Fanuc TP program (LS listing): HS_oV_wD.ls

/PROG  HS_oV_wD
/ATTR
COMMENT	= "18-08-10 08:42:27";
PROG_SIZE	= 0;
DEFAULT_GROUP	= 1, 1, *, *, *;
/APPL
    ARC Welding Equipment: 1, *, *, *, *;
/MN
   1:  CALL HOME_ALL;
   1:  UFRAME_NUM = 1;
   1:  UTOOL_NUM = 3;
   1:  COL GUARD ADJUST 150;
   1:  PR[91] = PR[90];
   1:! Sicherheitspunkt;
   1:  PR[92] = PR[90];
   1:  PR[92] = PR[GP1:92,3] + 50;
   1:J PR[92];
   1:  PR[GP1:91,1] = PR[GP1:90,1] + -0.150;
   1:  PR[GP1:91,2] = PR[GP1:90,2] + 0.396;
   1:  PR[GP1:91,3] = PR[GP1:90,3] + 1.330;
   1:L PR[91] 10mm/sec CNT100;
   1:  PR[GP1:91,1] = PR[GP1:90,1] + -3.720;
   1:  PR[GP1:91,2] = PR[GP1:90,2] + 1.719;
   1:L PR[91] 10mm/sec CNT100;
   1:  PR[GP1:91,1] = PR[GP1:90,1] + -5.535;
   1:  PR[GP1:91,2] = PR[GP1:90,2] + 4.999;
   1:L PR[91] 10mm/sec CNT100;
   1:  PR[GP1:91,1] = PR[GP1:90,1] + -9.508;
   1:  PR[GP1:91,2] = PR[GP1:90,2] + 16.323;
   1:L PR[91] 10mm/sec CNT100;
   1:  PR[GP1:91,1] = PR[GP1:90,1] + -9.633;
   1:  PR[GP1:91,2] = PR[GP1:90,2] + 16.823;
   1:L PR[91] 10mm/sec CNT100;
   1:  PR[GP1:91,1] = PR[GP1:90,1] + -9.801;
   1:  PR[GP1:91,2] = PR[GP1:90,2] + 17.188;
   1:L PR[91] 10mm/sec CNT100;
   1:  PR[GP1:91,1] = PR[GP1:90,1] + -17.552;
   1:  PR[GP1:91,2] = PR[GP1:90,2] + 26.184;
   1:L PR[91] 10mm/sec CNT100;
   1:  PR[GP1:91,1] = PR[GP1:90,1] + -17.850;
   1:  PR[GP1:91,2] = PR[GP1:90,2] + 26.604;
   1:L PR[91] 10mm/sec CNT100;
   1:  PR[GP1:91,1] = PR[GP1:90,1] + -18.140;
   1:  PR[GP1:91,2] = PR[GP1:90,2] + 26.882;
   1:L PR[91] 10mm/sec CNT100;
   1:  PR[GP1:91,1] = PR[GP1:90,1] + -28.635;
   1:  PR[GP1:91,2] = PR[GP1:90,2] + 32.423;
   1:L PR[91] 10mm/sec CNT100;
   1:  PR[GP1:91,1] = PR[GP1:90,1] + -29.066;
   1:  PR[GP1:91,2] = PR[GP1:90,2] + 32.704;
   1:L PR[91] 10mm/sec CNT100;
   1:  PR[GP1:91,1] = PR[GP1:90,1] + -29.438;
   1:  PR[GP1:91,2] = PR[GP1:90,2] + 32.858;
   1:L PR[91] 10mm/sec CNT100;
   1:  PR[GP1:91,1] = PR[GP1:90,1] + -41.237;
   1:  PR[GP1:91,2] = PR[GP1:90,2] + 34.183;
   1:L PR[91] 10mm/sec CNT100;
   1:  PR[GP1:91,1] = PR[GP1:90,1] + -41.741;
   1:  PR[GP1:91,2] = PR[GP1:90,2] + 34.288;
   1:L PR[91] 10mm/sec CNT100;
   1:  PR[GP1:91,1] = PR[GP1:90,1] + -42.143;
   1:  PR[GP1:91,2] = PR[GP1:90,2] + 34.295;
   1:L PR[91] 10mm/sec CNT100;
   1:  PR[GP1:91,1] = PR[GP1:90,1] + -53.611;
   1:  PR[GP1:91,2] = PR[GP1:90,2] + 31.219;
   1:L PR[91] 10mm/sec CNT100;
   1:  PR[GP1:91,1] = PR[GP1:90,1] + -54.119;
   1:  PR[GP1:91,2] = PR[GP1:90,2] + 31.132;
   1:L PR[91] 10mm/sec CNT100;
   1:  PR[GP1:91,1] = PR[GP1:90,1] + -54.496;
   1:  PR[GP1:91,2] = PR[GP1:90,2] + 30.992;
   1:L PR[91] 10mm/sec CNT100;
   1:  PR[GP1:91,1] = PR[GP1:90,1] + -64.044;
   1:  PR[GP1:91,2] = PR[GP1:90,2] + 23.943;
   1:L PR[91] 10mm/sec CNT100;
   1:  PR[GP1:91,1] = PR[GP1:90,1] + -64.485;
   1:  PR[GP1:91,2] = PR[GP1:90,2] + 23.677;
   1:L PR[91] 10mm/sec CNT100;
   1:  PR[GP1:91,1] = PR[GP1:90,1] + -64.785;
   1:  PR[GP1:91,2] = PR[GP1:90,2] + 23.409;
   1:L PR[91] 10mm/sec CNT100;
   1:  PR[GP1:91,1] = PR[GP1:90,1] + -71.103;
   1:  PR[GP1:91,2] = PR[GP1:90,2] + 13.353;
   1:L PR[91] 10mm/sec CNT100;
   1:  PR[GP1:91,1] = PR[GP1:90,1] + -71.416;
   1:  PR[GP1:91,2] = PR[GP1:90,2] + 12.944;
   1:L PR[91] 10mm/sec CNT100;
   1:  PR[GP1:91,1] = PR[GP1:90,1] + -71.597;
   1:  PR[GP1:91,2] = PR[GP1:90,2] + 12.585;
   1:L PR[91] 10mm/sec CNT100;
   1:  PR[GP1:91,1] = PR[GP1:90,1] + -73.804;
   1:  PR[GP1:91,2] = PR[GP1:90,2] + 0.919;
   1:L PR[91] 10mm/sec CNT100;
   1:  PR[GP1:91,1] = PR[GP1:90,1] + -73.947;
   1:  PR[GP1:91,2] = PR[GP1:90,2] + 0.424;
   1:L PR[91] 10mm/sec CNT100;
   1:  PR[GP1:91,1] = PR[GP1:90,1] + -73.984;
   1:  PR[GP1:91,2] = PR[GP1:90,2] + 0.024;
   1:L PR[91] 10mm/sec CNT100;
   1:  PR[GP1:91,1] = PR[GP1:90,1] + -71.777;
   1:  PR[GP1:91,2] = PR[GP1:90,2] + -11.642;
   1:L PR[91] 10mm/sec CNT100;
   1:  PR[GP1:91,1] = PR[GP1:90,1] + -71.729;
   1:  PR[GP1:91,2] = PR[GP1:90,2] + -12.155;
   1:L PR[91] 10mm/sec CNT100;
   1:  PR[GP1:91,1] = PR[GP1:90,1] + -71.610;
   1:  PR[GP1:91,2] = PR[GP1:90,2] + -12.569;
   1:L PR[91] 10mm/sec CNT100;
   1:  PR[GP1:91,1] = PR[GP1:90,1] + -71.403;
   1:  PR[GP1:91,2] = PR[GP1:90,2] + -12.978;
   1:L PR[91] 10mm/sec CNT100;
   1:  PR[GP1:91,1] = PR[GP1:90,1] + -65.085;
   1:  PR[GP1:91,2] = PR[GP1:90,2] + -23.035;
   1:L PR[91] 10mm/sec CNT100;
   1:  PR[GP1:91,1] = PR[GP1:90,1] + -64.806;
   1:  PR[GP1:91,2] = PR[GP1:90,2] + -23.399;
   1:L PR[91] 10mm/sec CNT100;
   1:  PR[GP1:91,1] = PR[GP1:90,1] + -64.464;
   1:  PR[GP1:91,2] = PR[GP1:90,2] + -23.705;
   1:L PR[91] 10mm/sec CNT100;
   1:  PR[GP1:91,1] = PR[GP1:90,1] + -54.915;
   1:  PR[GP1:91,2] = PR[GP1:90,2] + -30.754;
   1:L PR[91] 10mm/sec CNT100;
   1:  PR[GP1:91,1] = PR[GP1:90,1] + -54.522;
   1:  PR[GP1:91,2] = PR[GP1:90,2] + -30.991;
   1:L PR[91] 10mm/sec CNT100;
   1:  PR[GP1:91,1] = PR[GP1:90,1] + -54.092;
   1:  PR[GP1:91,2] = PR[GP1:90,2] + -31.151;
   1:L PR[91] 10mm/sec CNT100;
   1:  PR[GP1:91,1] = PR[GP1:90,1] + -42.624;
   1:  PR[GP1:91,2] = PR[GP1:90,2] + -34.227;
   1:L PR[91] 10mm/sec CNT100;
   1:  PR[GP1:91,1] = PR[GP1:90,1] + -42.171;
   1:  PR[GP1:91,2] = PR[GP1:90,2] + -34.304;
   1:L PR[91] 10mm/sec CNT100;
   1:  PR[GP1:91,1] = PR[GP1:90,1] + -41.713;
   1:  PR[GP1:91,2] = PR[GP1:90,2] + -34.296;
   1:L PR[91] 10mm/sec CNT100;
   1:  PR[GP1:91,1] = PR[GP1:90,1] + -29.913;
   1:  PR[GP1:91,2] = PR[GP1:90,2] + -32.971;
   1:L PR[91] 10mm/sec CNT100;
   1:  PR[GP1:91,1] = PR[GP1:90,1] + -29.464;
   1:  PR[GP1:91,2] = PR[GP1:90,2] + -32.878;
   1:L PR[91] 10mm/sec CNT100;
   1:  PR[GP1:91,1] = PR[GP1:90,1] + -29.040;
   1:  PR[GP1:91,2] = PR[GP1:90,2] + -32.702;
   1:L PR[91] 10mm/sec CNT100;
   1:  PR[GP1:91,1] = PR[GP1:90,1] + -18.545;
   1:  PR[GP1:91,2] = PR[GP1:90,2] + -27.162;
   1:L PR[91] 10mm/sec CNT100;
   1:  PR[GP1:91,1] = PR[GP1:90,1] + -18.161;
   1:  PR[GP1:91,2] = PR[GP1:90,2] + -26.911;
   1:L PR[91] 10mm/sec CNT100;
   1:  PR[GP1:91,1] = PR[GP1:90,1] + -17.830;
   1:  PR[GP1:91,2] = PR[GP1:90,2] + -26.593;
   1:L PR[91] 10mm/sec CNT100;
   1:  PR[GP1:91,1] = PR[GP1:90,1] + -10.079;
   1:  PR[GP1:91,2] = PR[GP1:90,2] + -17.597;
   1:L PR[91] 10mm/sec CNT100;
   1:  PR[GP1:91,1] = PR[GP1:90,1] + -9.813;
   1:  PR[GP1:91,2] = PR[GP1:90,2] + -17.223;
   1:L PR[91] 10mm/sec CNT100;
   1:  PR[GP1:91,1] = PR[GP1:90,1] + -9.621;
   1:  PR[GP1:91,2] = PR[GP1:90,2] + -16.806;
   1:L PR[91] 10mm/sec CNT100;
   1:  PR[GP1:91,1] = PR[GP1:90,1] + -5.692;
   1:  PR[GP1:91,2] = PR[GP1:90,2] + -5.609;
   1:L PR[91] 10mm/sec CNT100;
   1:  PR[GP1:91,1] = PR[GP1:90,1] + -5.549;
   1:  PR[GP1:91,2] = PR[GP1:90,2] + -5.033;
   1:L PR[91] 10mm/sec CNT100;
   1:  PR[GP1:91,1] = PR[GP1:90,1] + -3.720;
   1:  PR[GP1:91,2] = PR[GP1:90,2] + -1.728;
   1:L PR[91] 10mm/sec CNT100;
   1:  PR[GP1:91,1] = PR[GP1:90,1] + -0.150;
   1:  PR[GP1:91,2] = PR[GP1:90,2] + -0.404;
   1:L PR[91] 10mm/sec CNT100;
   1:  PR[GP1:91,1] = PR[GP1:90,1] + 0.971;
   1:L PR[91] 10mm/sec CNT100;
   1:  PR[GP1:91,1] = PR[GP1:90,1] + 4.540;
   1:  PR[GP1:91,2] = PR[GP1:90,2] + -1.728;
   1:L PR[91] 10mm/sec CNT100;
   1:  PR[GP1:91,1] = PR[GP1:90,1] + 6.356;
   1:  PR[GP1:91,2] = PR[GP1:90,2] + -5.008;
   1:L PR[91] 10mm/sec CNT100;
   1:  PR[GP1:91,1] = PR[GP1:90,1] + 10.329;
   1:  PR[GP1:91,2] = PR[GP1:90,2] + -16.332;
   1:L PR[91] 10mm/sec CNT100;
   1:  PR[GP1:91,1] = PR[GP1:90,1] + 10.453;
   1:  PR[GP1:91,2] = PR[GP1:90,2] + -16.832;
   1:L PR[91] 10mm/sec CNT100;
   1:  PR[GP1:91,1] = PR[GP1:90,1] + 10.621;
   1:  PR[GP1:91,2] = PR[GP1:90,2] + -17.197;
   1:L PR[91] 10mm/sec CNT100;
   1:  PR[GP1:91,1] = PR[GP1:90,1] + 18.373;
   1:  PR[GP1:91,2] = PR[GP1:90,2] + -26.193;
   1:L PR[91] 10mm/sec CNT100;
   1:  PR[GP1:91,1] = PR[GP1:90,1] + 18.671;
   1:  PR[GP1:91,2] = PR[GP1:90,2] + -26.612;
   1:L PR[91] 10mm/sec CNT100;
   1:  PR[GP1:91,1] = PR[GP1:90,1] + 18.961;
   1:  PR[GP1:91,2] = PR[GP1:90,2] + -26.891;
   1:L PR[91] 10mm/sec CNT100;
   1:  PR[GP1:91,1] = PR[GP1:90,1] + 29.456;
   1:  PR[GP1:91,2] = PR[GP1:90,2] + -32.431;
   1:L PR[91] 10mm/sec CNT100;
   1:  PR[GP1:91,1] = PR[GP1:90,1] + 29.887;
   1:  PR[GP1:91,2] = PR[GP1:90,2] + -32.713;
   1:L PR[91] 10mm/sec CNT100;
   1:  PR[GP1:91,1] = PR[GP1:90,1] + 30.259;
   1:  PR[GP1:91,2] = PR[GP1:90,2] + -32.867;
   1:L PR[91] 10mm/sec CNT100;
   1:  PR[GP1:91,1] = PR[GP1:90,1] + 42.058;
   1:  PR[GP1:91,2] = PR[GP1:90,2] + -34.192;
   1:L PR[91] 10mm/sec CNT100;
   1:  PR[GP1:91,1] = PR[GP1:90,1] + 42.562;
   1:  PR[GP1:91,2] = PR[GP1:90,2] + -34.296;
   1:L PR[91] 10mm/sec CNT100;
   1:  PR[GP1:91,1] = PR[GP1:90,1] + 42.964;
   1:  PR[GP1:91,2] = PR[GP1:90,2] + -34.304;
   1:L PR[91] 10mm/sec CNT100;
   1:  PR[GP1:91,1] = PR[GP1:90,1] + 54.432;
   1:  PR[GP1:91,2] = PR[GP1:90,2] + -31.228;
   1:L PR[91] 10mm/sec CNT100;
   1:  PR[GP1:91,1] = PR[GP1:90,1] + 54.939;
   1:  PR[GP1:91,2] = PR[GP1:90,2] + -31.141;
   1:L PR[91] 10mm/sec CNT100;
   1:  PR[GP1:91,1] = PR[GP1:90,1] + 55.316;
   1:  PR[GP1:91,2] = PR[GP1:90,2] + -31.001;
   1:L PR[91] 10mm/sec CNT100;
   1:  PR[GP1:91,1] = PR[GP1:90,1] + 64.865;
   1:  PR[GP1:91,2] = PR[GP1:90,2] + -23.952;
   1:L PR[91] 10mm/sec CNT100;
   1:  PR[GP1:91,1] = PR[GP1:90,1] + 65.306;
   1:  PR[GP1:91,2] = PR[GP1:90,2] + -23.686;
   1:L PR[91] 10mm/sec CNT100;
   1:  PR[GP1:91,1] = PR[GP1:90,1] + 65.605;
   1:  PR[GP1:91,2] = PR[GP1:90,2] + -23.418;
   1:L PR[91] 10mm/sec CNT100;
   1:  PR[GP1:91,1] = PR[GP1:90,1] + 71.923;
   1:  PR[GP1:91,2] = PR[GP1:90,2] + -13.361;
   1:L PR[91] 10mm/sec CNT100;
   1:  PR[GP1:91,1] = PR[GP1:90,1] + 72.237;
   1:  PR[GP1:91,2] = PR[GP1:90,2] + -12.953;
   1:L PR[91] 10mm/sec CNT100;
   1:  PR[GP1:91,1] = PR[GP1:90,1] + 72.418;
   1:  PR[GP1:91,2] = PR[GP1:90,2] + -12.594;
   1:L PR[91] 10mm/sec CNT100;
   1:  PR[GP1:91,1] = PR[GP1:90,1] + 74.625;
   1:  PR[GP1:91,2] = PR[GP1:90,2] + -0.928;
   1:L PR[91] 10mm/sec CNT100;
   1:  PR[GP1:91,1] = PR[GP1:90,1] + 74.767;
   1:  PR[GP1:91,2] = PR[GP1:90,2] + -0.433;
   1:L PR[91] 10mm/sec CNT100;
   1:  PR[GP1:91,1] = PR[GP1:90,1] + 74.805;
   1:  PR[GP1:91,2] = PR[GP1:90,2] + -0.033;
   1:L PR[91] 10mm/sec CNT100;
   1:  PR[GP1:91,1] = PR[GP1:90,1] + 72.598;
   1:  PR[GP1:91,2] = PR[GP1:90,2] + 11.633;
   1:L PR[91] 10mm/sec CNT100;
   1:  PR[GP1:91,1] = PR[GP1:90,1] + 72.550;
   1:  PR[GP1:91,2] = PR[GP1:90,2] + 12.146;
   1:L PR[91] 10mm/sec CNT100;
   1:  PR[GP1:91,1] = PR[GP1:90,1] + 72.430;
   1:  PR[GP1:91,2] = PR[GP1:90,2] + 12.560;
   1:L PR[91] 10mm/sec CNT100;
   1:  PR[GP1:91,1] = PR[GP1:90,1] + 72.224;
   1:  PR[GP1:91,2] = PR[GP1:90,2] + 12.969;
   1:L PR[91] 10mm/sec CNT100;
   1:  PR[GP1:91,1] = PR[GP1:90,1] + 65.906;
   1:  PR[GP1:91,2] = PR[GP1:90,2] + 23.026;
   1:L PR[91] 10mm/sec CNT100;
   1:  PR[GP1:91,1] = PR[GP1:90,1] + 65.627;
   1:  PR[GP1:91,2] = PR[GP1:90,2] + 23.390;
   1:L PR[91] 10mm/sec CNT100;
   1:  PR[GP1:91,1] = PR[GP1:90,1] + 65.285;
   1:  PR[GP1:91,2] = PR[GP1:90,2] + 23.696;
   1:L PR[91] 10mm/sec CNT100;
   1:  PR[GP1:91,1] = PR[GP1:90,1] + 55.736;
   1:  PR[GP1:91,2] = PR[GP1:90,2] + 30.746;
   1:L PR[91] 10mm/sec CNT100;
   1:  PR[GP1:91,1] = PR[GP1:90,1] + 55.343;
   1:  PR[GP1:91,2] = PR[GP1:90,2] + 30.982;
   1:L PR[91] 10mm/sec CNT100;
   1:  PR[GP1:91,1] = PR[GP1:90,1] + 54.913;
   1:  PR[GP1:91,2] = PR[GP1:90,2] + 31.142;
   1:L PR[91] 10mm/sec CNT100;
   1:  PR[GP1:91,1] = PR[GP1:90,1] + 43.444;
   1:  PR[GP1:91,2] = PR[GP1:90,2] + 34.218;
   1:L PR[91] 10mm/sec CNT100;
   1:  PR[GP1:91,1] = PR[GP1:90,1] + 42.992;
   1:  PR[GP1:91,2] = PR[GP1:90,2] + 34.295;
   1:L PR[91] 10mm/sec CNT100;
   1:  PR[GP1:91,1] = PR[GP1:90,1] + 42.533;
   1:  PR[GP1:91,2] = PR[GP1:90,2] + 34.287;
   1:L PR[91] 10mm/sec CNT100;
   1:  PR[GP1:91,1] = PR[GP1:90,1] + 30.734;
   1:  PR[GP1:91,2] = PR[GP1:90,2] + 32.962;
   1:L PR[91] 10mm/sec CNT100;
   1:  PR[GP1:91,1] = PR[GP1:90,1] + 30.285;
   1:  PR[GP1:91,2] = PR[GP1:90,2] + 32.869;
   1:L PR[91] 10mm/sec CNT100;
   1:  PR[GP1:91,1] = PR[GP1:90,1] + 29.861;
   1:  PR[GP1:91,2] = PR[GP1:90,2] + 32.694;
   1:L PR[91] 10mm/sec CNT100;
   1:  PR[GP1:91,1] = PR[GP1:90,1] + 19.365;
   1:  PR[GP1:91,2] = PR[GP1:90,2] + 27.153;
   1:L PR[91] 10mm/sec CNT100;
   1:  PR[GP1:91,1] = PR[GP1:90,1] + 18.981;
   1:  PR[GP1:91,2] = PR[GP1:90,2] + 26.902;
   1:L PR[91] 10mm/sec CNT100;
   1:  PR[GP1:91,1] = PR[GP1:90,1] + 18.651;
   1:  PR[GP1:91,2] = PR[GP1:90,2] + 26.584;
   1:L PR[91] 10mm/sec CNT100;
   1:  PR[GP1:91,1] = PR[GP1:90,1] + 10.899;
   1:  PR[GP1:91,2] = PR[GP1:90,2] + 17.588;
   1:L PR[91] 10mm/sec CNT100;
   1:  PR[GP1:91,1] = PR[GP1:90,1] + 10.633;
   1:  PR[GP1:91,2] = PR[GP1:90,2] + 17.214;
   1:L PR[91] 10mm/sec CNT100;
   1:  PR[GP1:91,1] = PR[GP1:90,1] + 10.442;
   1:  PR[GP1:91,2] = PR[GP1:90,2] + 16.797;
   1:L PR[91] 10mm/sec CNT100;
   1:  PR[GP1:91,1] = PR[GP1:90,1] + 6.513;
   1:  PR[GP1:91,2] = PR[GP1:90,2] + 5.600;
   1:L PR[91] 10mm/sec CNT100;
   1:  PR[GP1:91,1] = PR[GP1:90,1] + 6.369;
   1:  PR[GP1:91,2] = PR[GP1:90,2] + 5.024;
   1:L PR[91] 10mm/sec CNT100;
   1:  PR[GP1:91,1] = PR[GP1:90,1] + 4.540;
   1:  PR[GP1:91,2] = PR[GP1:90,2] + 1.719;
   1:L PR[91] 10mm/sec CNT100;
   1:  PR[GP1:91,1] = PR[GP1:90,1] + 0.971;
   1:  PR[GP1:91,2] = PR[GP1:90,2] + 0.396;
   1:L PR[91] 10mm/sec CNT100;
   1:  PR[GP1:91,1] = PR[GP1:90,1] + -0.150;
   1:L PR[91] 10mm/sec CNT100;
   1:  PR[GP1:91,1] = PR[GP1:90,1] + -3.720;
   1:  PR[GP1:91,2] = PR[GP1:90,2] + 1.719;
   1:  PR[GP1:91,3] = PR[GP1:90,3] + 2.660;
   1:L PR[91] 10mm/sec CNT100;
   1:  PR[GP1:91,1] = PR[GP1:90,1] + -5.535;
   1:  PR[GP1:91,2] = PR[GP1:90,2] + 4.999;
   1:L PR[91] 10mm/sec CNT100;
   1:  PR[GP1:91,1] = PR[GP1:90,1] + -8.793;
   1:  PR[GP1:91,2] = PR[GP1:90,2] + 14.283;
   1:L PR[91] 10mm/sec CNT100;
   1:  PR[GP1:91,1] = PR[GP1:90,1] + -9.180;
   1:  PR[GP1:91,2] = PR[GP1:90,2] + 15.837;
   1:L PR[91] 10mm/sec CNT100;
   1:  PR[GP1:91,1] = PR[GP1:90,1] + -9.801;
   1:  PR[GP1:91,2] = PR[GP1:90,2] + 17.189;
   1:L PR[91] 10mm/sec CNT100;
   1:  PR[GP1:91,1] = PR[GP1:90,1] + -16.140;
   1:  PR[GP1:91,2] = PR[GP1:90,2] + 24.546;
   1:L PR[91] 10mm/sec CNT100;
   1:  PR[GP1:91,1] = PR[GP1:90,1] + -17.068;
   1:  PR[GP1:91,2] = PR[GP1:90,2] + 25.851;
   1:L PR[91] 10mm/sec CNT100;
   1:  PR[GP1:91,1] = PR[GP1:90,1] + -18.141;
   1:  PR[GP1:91,2] = PR[GP1:90,2] + 26.883;
   1:L PR[91] 10mm/sec CNT100;
   1:  PR[GP1:91,1] = PR[GP1:90,1] + -26.724;
   1:  PR[GP1:91,2] = PR[GP1:90,2] + 31.414;
   1:L PR[91] 10mm/sec CNT100;
   1:  PR[GP1:91,1] = PR[GP1:90,1] + -28.064;
   1:  PR[GP1:91,2] = PR[GP1:90,2] + 32.290;
   1:L PR[91] 10mm/sec CNT100;
   1:  PR[GP1:91,1] = PR[GP1:90,1] + -29.439;
   1:  PR[GP1:91,2] = PR[GP1:90,2] + 32.858;
   1:L PR[91] 10mm/sec CNT100;
   1:  PR[GP1:91,1] = PR[GP1:90,1] + -39.088;
   1:  PR[GP1:91,2] = PR[GP1:90,2] + 33.942;
   1:L PR[91] 10mm/sec CNT100;
   1:  PR[GP1:91,1] = PR[GP1:90,1] + -40.656;
   1:  PR[GP1:91,2] = PR[GP1:90,2] + 34.268;
   1:L PR[91] 10mm/sec CNT100;
   1:  PR[GP1:91,1] = PR[GP1:90,1] + -42.144;
   1:  PR[GP1:91,2] = PR[GP1:90,2] + 34.295;
   1:L PR[91] 10mm/sec CNT100;
   1:  PR[GP1:91,1] = PR[GP1:90,1] + -51.523;
   1:  PR[GP1:91,2] = PR[GP1:90,2] + 31.779;
   1:L PR[91] 10mm/sec CNT100;
   1:  PR[GP1:91,1] = PR[GP1:90,1] + -53.101;
   1:  PR[GP1:91,2] = PR[GP1:90,2] + 31.510;
   1:L PR[91] 10mm/sec CNT100;
   1:  PR[GP1:91,1] = PR[GP1:90,1] + -54.496;
   1:  PR[GP1:91,2] = PR[GP1:90,2] + 30.992;
   1:L PR[91] 10mm/sec CNT100;
   1:  PR[GP1:91,1] = PR[GP1:90,1] + -62.305;
   1:  PR[GP1:91,2] = PR[GP1:90,2] + 25.227;
   1:L PR[91] 10mm/sec CNT100;
   1:  PR[GP1:91,1] = PR[GP1:90,1] + -63.676;
   1:  PR[GP1:91,2] = PR[GP1:90,2] + 24.400;
   1:L PR[91] 10mm/sec CNT100;
   1:  PR[GP1:91,1] = PR[GP1:90,1] + -64.786;
   1:  PR[GP1:91,2] = PR[GP1:90,2] + 23.408;
   1:L PR[91] 10mm/sec CNT100;
   1:  PR[GP1:91,1] = PR[GP1:90,1] + -69.952;
   1:  PR[GP1:91,2] = PR[GP1:90,2] + 15.184;
   1:L PR[91] 10mm/sec CNT100;
   1:  PR[GP1:91,1] = PR[GP1:90,1] + -70.927;
   1:  PR[GP1:91,2] = PR[GP1:90,2] + 13.914;
   1:L PR[91] 10mm/sec CNT100;
   1:  PR[GP1:91,1] = PR[GP1:90,1] + -71.597;
   1:  PR[GP1:91,2] = PR[GP1:90,2] + 12.585;
   1:L PR[91] 10mm/sec CNT100;
   1:  PR[GP1:91,1] = PR[GP1:90,1] + -73.402;
   1:  PR[GP1:91,2] = PR[GP1:90,2] + 3.044;
   1:L PR[91] 10mm/sec CNT100;
   1:  PR[GP1:91,1] = PR[GP1:90,1] + -73.845;
   1:  PR[GP1:91,2] = PR[GP1:90,2] + 1.506;
   1:L PR[91] 10mm/sec CNT100;
   1:  PR[GP1:91,1] = PR[GP1:90,1] + -73.984;
   1:  PR[GP1:91,2] = PR[GP1:90,2] + 0.024;
   1:L PR[91] 10mm/sec CNT100;
   1:  PR[GP1:91,1] = PR[GP1:90,1] + -72.179;
   1:  PR[GP1:91,2] = PR[GP1:90,2] + -9.517;
   1:L PR[91] 10mm/sec CNT100;
   1:  PR[GP1:91,1] = PR[GP1:90,1] + -72.030;
   1:  PR[GP1:91,2] = PR[GP1:90,2] + -11.111;
   1:L PR[91] 10mm/sec CNT100;
   1:  PR[GP1:91,1] = PR[GP1:90,1] + -71.610;
   1:  PR[GP1:91,2] = PR[GP1:90,2] + -12.568;
   1:L PR[91] 10mm/sec CNT100;
   1:  PR[GP1:91,1] = PR[GP1:90,1] + -70.914;
   1:  PR[GP1:91,2] = PR[GP1:90,2] + -13.948;
   1:L PR[91] 10mm/sec CNT100;
   1:  PR[GP1:91,1] = PR[GP1:90,1] + -65.747;
   1:  PR[GP1:91,2] = PR[GP1:90,2] + -22.172;
   1:L PR[91] 10mm/sec CNT100;
   1:  PR[GP1:91,1] = PR[GP1:90,1] + -64.807;
   1:  PR[GP1:91,2] = PR[GP1:90,2] + -23.398;
   1:L PR[91] 10mm/sec CNT100;
   1:  PR[GP1:91,1] = PR[GP1:90,1] + -63.655;
   1:  PR[GP1:91,2] = PR[GP1:90,2] + -24.428;
   1:L PR[91] 10mm/sec CNT100;
   1:  PR[GP1:91,1] = PR[GP1:90,1] + -55.846;
   1:  PR[GP1:91,2] = PR[GP1:90,2] + -30.193;
   1:L PR[91] 10mm/sec CNT100;
   1:  PR[GP1:91,1] = PR[GP1:90,1] + -54.523;
   1:  PR[GP1:91,2] = PR[GP1:90,2] + -30.991;
   1:L PR[91] 10mm/sec CNT100;
   1:  PR[GP1:91,1] = PR[GP1:90,1] + -53.075;
   1:  PR[GP1:91,2] = PR[GP1:90,2] + -31.529;
   1:L PR[91] 10mm/sec CNT100;
   1:  PR[GP1:91,1] = PR[GP1:90,1] + -43.695;
   1:  PR[GP1:91,2] = PR[GP1:90,2] + -34.045;
   1:L PR[91] 10mm/sec CNT100;
   1:  PR[GP1:91,1] = PR[GP1:90,1] + -42.172;
   1:  PR[GP1:91,2] = PR[GP1:90,2] + -34.304;
   1:L PR[91] 10mm/sec CNT100;
   1:  PR[GP1:91,1] = PR[GP1:90,1] + -40.628;
   1:  PR[GP1:91,2] = PR[GP1:90,2] + -34.276;
   1:L PR[91] 10mm/sec CNT100;
   1:  PR[GP1:91,1] = PR[GP1:90,1] + -30.978;
   1:  PR[GP1:91,2] = PR[GP1:90,2] + -33.193;
   1:L PR[91] 10mm/sec CNT100;
   1:  PR[GP1:91,1] = PR[GP1:90,1] + -29.465;
   1:  PR[GP1:91,2] = PR[GP1:90,2] + -32.878;
   1:L PR[91] 10mm/sec CNT100;
   1:  PR[GP1:91,1] = PR[GP1:90,1] + -28.038;
   1:  PR[GP1:91,2] = PR[GP1:90,2] + -32.288;
   1:L PR[91] 10mm/sec CNT100;
   1:  PR[GP1:91,1] = PR[GP1:90,1] + -19.454;
   1:  PR[GP1:91,2] = PR[GP1:90,2] + -27.757;
   1:L PR[91] 10mm/sec CNT100;
   1:  PR[GP1:91,1] = PR[GP1:90,1] + -18.161;
   1:  PR[GP1:91,2] = PR[GP1:90,2] + -26.911;
   1:L PR[91] 10mm/sec CNT100;
   1:  PR[GP1:91,1] = PR[GP1:90,1] + -17.048;
   1:  PR[GP1:91,2] = PR[GP1:90,2] + -25.840;
   1:L PR[91] 10mm/sec CNT100;
   1:  PR[GP1:91,1] = PR[GP1:90,1] + -10.708;
   1:  PR[GP1:91,2] = PR[GP1:90,2] + -18.483;
   1:L PR[91] 10mm/sec CNT100;
   1:  PR[GP1:91,1] = PR[GP1:90,1] + -9.813;
   1:  PR[GP1:91,2] = PR[GP1:90,2] + -17.224;
   1:L PR[91] 10mm/sec CNT100;
   1:  PR[GP1:91,1] = PR[GP1:90,1] + -9.168;
   1:  PR[GP1:91,2] = PR[GP1:90,2] + -15.820;
   1:L PR[91] 10mm/sec CNT100;
   1:  PR[GP1:91,1] = PR[GP1:90,1] + -5.955;
   1:  PR[GP1:91,2] = PR[GP1:90,2] + -6.663;
   1:L PR[91] 10mm/sec CNT100;
   1:  PR[GP1:91,1] = PR[GP1:90,1] + -5.549;
   1:  PR[GP1:91,2] = PR[GP1:90,2] + -5.033;
   1:L PR[91] 10mm/sec CNT100;
   1:  PR[GP1:91,1] = PR[GP1:90,1] + -3.720;
   1:  PR[GP1:91,2] = PR[GP1:90,2] + -1.728;
   1:L PR[91] 10mm/sec CNT100;
   1:  PR[GP1:91,1] = PR[GP1:90,1] + -0.150;
   1:  PR[GP1:91,2] = PR[GP1:90,2] + -0.404;
   1:L PR[91] 10mm/sec CNT100;
   1:  PR[GP1:91,1] = PR[GP1:90,1] + 0.971;
   1:L PR[91] 10mm/sec CNT100;
   1:  PR[GP1:91,1] = PR[GP1:90,1] + 4.540;
   1:  PR[GP1:91,2] = PR[GP1:90,2] + -1.728;
   1:L PR[91] 10mm/sec CNT100;
   1:  PR[GP1:91,1] = PR[GP1:90,1] + 6.356;
   1:  PR[GP1:91,2] = PR[GP1:90,2] + -5.008;
   1:L PR[91] 10mm/sec CNT100;
   1:  PR[GP1:91,1] = PR[GP1:90,1] + 9.613;
   1:  PR[GP1:91,2] = PR[GP1:90,2] + -14.292;
   1:L PR[91] 10mm/sec CNT100;
   1:  PR[GP1:91,1] = PR[GP1:90,1] + 10.000;
   1:  PR[GP1:91,2] = PR[GP1:90,2] + -15.846;
   1:L PR[91] 10mm/sec CNT100;
   1:  PR[GP1:91,1] = PR[GP1:90,1] + 10.622;
   1:  PR[GP1:91,2] = PR[GP1:90,2] + -17.198;
   1:L PR[91] 10mm/sec CNT100;
   1:  PR[GP1:91,1] = PR[GP1:90,1] + 16.961;
   1:  PR[GP1:91,2] = PR[GP1:90,2] + -24.555;
   1:L PR[91] 10mm/sec CNT100;
   1:  PR[GP1:91,1] = PR[GP1:90,1] + 17.889;
   1:  PR[GP1:91,2] = PR[GP1:90,2] + -25.860;
   1:L PR[91] 10mm/sec CNT100;
   1:  PR[GP1:91,1] = PR[GP1:90,1] + 18.961;
   1:  PR[GP1:91,2] = PR[GP1:90,2] + -26.892;
   1:L PR[91] 10mm/sec CNT100;
   1:  PR[GP1:91,1] = PR[GP1:90,1] + 27.544;
   1:  PR[GP1:91,2] = PR[GP1:90,2] + -31.422;
   1:L PR[91] 10mm/sec CNT100;
   1:  PR[GP1:91,1] = PR[GP1:90,1] + 28.884;
   1:  PR[GP1:91,2] = PR[GP1:90,2] + -32.298;
   1:L PR[91] 10mm/sec CNT100;
   1:  PR[GP1:91,1] = PR[GP1:90,1] + 30.260;
   1:  PR[GP1:91,2] = PR[GP1:90,2] + -32.867;
   1:L PR[91] 10mm/sec CNT100;
   1:  PR[GP1:91,1] = PR[GP1:90,1] + 39.909;
   1:  PR[GP1:91,2] = PR[GP1:90,2] + -33.951;
   1:L PR[91] 10mm/sec CNT100;
   1:  PR[GP1:91,1] = PR[GP1:90,1] + 41.477;
   1:  PR[GP1:91,2] = PR[GP1:90,2] + -34.277;
   1:L PR[91] 10mm/sec CNT100;
   1:  PR[GP1:91,1] = PR[GP1:90,1] + 42.965;
   1:  PR[GP1:91,2] = PR[GP1:90,2] + -34.304;
   1:L PR[91] 10mm/sec CNT100;
   1:  PR[GP1:91,1] = PR[GP1:90,1] + 52.343;
   1:  PR[GP1:91,2] = PR[GP1:90,2] + -31.788;
   1:L PR[91] 10mm/sec CNT100;
   1:  PR[GP1:91,1] = PR[GP1:90,1] + 53.922;
   1:  PR[GP1:91,2] = PR[GP1:90,2] + -31.519;
   1:L PR[91] 10mm/sec CNT100;
   1:  PR[GP1:91,1] = PR[GP1:90,1] + 55.317;
   1:  PR[GP1:91,2] = PR[GP1:90,2] + -31.001;
   1:L PR[91] 10mm/sec CNT100;
   1:  PR[GP1:91,1] = PR[GP1:90,1] + 63.126;
   1:  PR[GP1:91,2] = PR[GP1:90,2] + -25.236;
   1:L PR[91] 10mm/sec CNT100;
   1:  PR[GP1:91,1] = PR[GP1:90,1] + 64.497;
   1:  PR[GP1:91,2] = PR[GP1:90,2] + -24.409;
   1:L PR[91] 10mm/sec CNT100;
   1:  PR[GP1:91,1] = PR[GP1:90,1] + 65.606;
   1:  PR[GP1:91,2] = PR[GP1:90,2] + -23.417;
   1:L PR[91] 10mm/sec CNT100;
   1:  PR[GP1:91,1] = PR[GP1:90,1] + 70.773;
   1:  PR[GP1:91,2] = PR[GP1:90,2] + -15.193;
   1:L PR[91] 10mm/sec CNT100;
   1:  PR[GP1:91,1] = PR[GP1:90,1] + 71.747;
   1:  PR[GP1:91,2] = PR[GP1:90,2] + -13.922;
   1:L PR[91] 10mm/sec CNT100;
   1:  PR[GP1:91,1] = PR[GP1:90,1] + 72.418;
   1:  PR[GP1:91,2] = PR[GP1:90,2] + -12.594;
   1:L PR[91] 10mm/sec CNT100;
   1:  PR[GP1:91,1] = PR[GP1:90,1] + 74.223;
   1:  PR[GP1:91,2] = PR[GP1:90,2] + -3.053;
   1:L PR[91] 10mm/sec CNT100;
   1:  PR[GP1:91,1] = PR[GP1:90,1] + 74.666;
   1:  PR[GP1:91,2] = PR[GP1:90,2] + -1.515;
   1:L PR[91] 10mm/sec CNT100;
   1:  PR[GP1:91,1] = PR[GP1:90,1] + 74.805;
   1:  PR[GP1:91,2] = PR[GP1:90,2] + -0.033;
   1:L PR[91] 10mm/sec CNT100;
   1:  PR[GP1:91,1] = PR[GP1:90,1] + 73.000;
   1:  PR[GP1:91,2] = PR[GP1:90,2] + 9.508;
   1:L PR[91] 10mm/sec CNT100;
   1:  PR[GP1:91,1] = PR[GP1:90,1] + 72.850;
   1:  PR[GP1:91,2] = PR[GP1:90,2] + 11.102;
   1:L PR[91] 10mm/sec CNT100;
   1:  PR[GP1:91,1] = PR[GP1:90,1] + 72.431;
   1:  PR[GP1:91,2] = PR[GP1:90,2] + 12.559;
   1:L PR[91] 10mm/sec CNT100;
   1:  PR[GP1:91,1] = PR[GP1:90,1] + 71.735;
   1:  PR[GP1:91,2] = PR[GP1:90,2] + 13.939;
   1:L PR[91] 10mm/sec CNT100;
   1:  PR[GP1:91,1] = PR[GP1:90,1] + 66.568;
   1:  PR[GP1:91,2] = PR[GP1:90,2] + 22.163;
   1:L PR[91] 10mm/sec CNT100;
   1:  PR[GP1:91,1] = PR[GP1:90,1] + 65.627;
   1:  PR[GP1:91,2] = PR[GP1:90,2] + 23.389;
   1:L PR[91] 10mm/sec CNT100;
   1:  PR[GP1:91,1] = PR[GP1:90,1] + 64.476;
   1:  PR[GP1:91,2] = PR[GP1:90,2] + 24.419;
   1:L PR[91] 10mm/sec CNT100;
   1:  PR[GP1:91,1] = PR[GP1:90,1] + 56.666;
   1:  PR[GP1:91,2] = PR[GP1:90,2] + 30.184;
   1:L PR[91] 10mm/sec CNT100;
   1:  PR[GP1:91,1] = PR[GP1:90,1] + 55.343;
   1:  PR[GP1:91,2] = PR[GP1:90,2] + 30.982;
   1:L PR[91] 10mm/sec CNT100;
   1:  PR[GP1:91,1] = PR[GP1:90,1] + 53.895;
   1:  PR[GP1:91,2] = PR[GP1:90,2] + 31.520;
   1:L PR[91] 10mm/sec CNT100;
   1:  PR[GP1:91,1] = PR[GP1:90,1] + 44.516;
   1:  PR[GP1:91,2] = PR[GP1:90,2] + 34.036;
   1:L PR[91] 10mm/sec CNT100;
   1:  PR[GP1:91,1] = PR[GP1:90,1] + 42.993;
   1:  PR[GP1:91,2] = PR[GP1:90,2] + 34.295;
   1:L PR[91] 10mm/sec CNT100;
   1:  PR[GP1:91,1] = PR[GP1:90,1] + 41.448;
   1:  PR[GP1:91,2] = PR[GP1:90,2] + 34.267;
   1:L PR[91] 10mm/sec CNT100;
   1:  PR[GP1:91,1] = PR[GP1:90,1] + 31.799;
   1:  PR[GP1:91,2] = PR[GP1:90,2] + 33.184;
   1:L PR[91] 10mm/sec CNT100;
   1:  PR[GP1:91,1] = PR[GP1:90,1] + 30.286;
   1:  PR[GP1:91,2] = PR[GP1:90,2] + 32.869;
   1:L PR[91] 10mm/sec CNT100;
   1:  PR[GP1:91,1] = PR[GP1:90,1] + 28.858;
   1:  PR[GP1:91,2] = PR[GP1:90,2] + 32.279;
   1:L PR[91] 10mm/sec CNT100;
   1:  PR[GP1:91,1] = PR[GP1:90,1] + 20.275;
   1:  PR[GP1:91,2] = PR[GP1:90,2] + 27.748;
   1:L PR[91] 10mm/sec CNT100;
   1:  PR[GP1:91,1] = PR[GP1:90,1] + 18.982;
   1:  PR[GP1:91,2] = PR[GP1:90,2] + 26.902;
   1:L PR[91] 10mm/sec CNT100;
   1:  PR[GP1:91,1] = PR[GP1:90,1] + 17.868;
   1:  PR[GP1:91,2] = PR[GP1:90,2] + 25.831;
   1:L PR[91] 10mm/sec CNT100;
   1:  PR[GP1:91,1] = PR[GP1:90,1] + 11.529;
   1:  PR[GP1:91,2] = PR[GP1:90,2] + 18.474;
   1:L PR[91] 10mm/sec CNT100;
   1:  PR[GP1:91,1] = PR[GP1:90,1] + 10.634;
   1:  PR[GP1:91,2] = PR[GP1:90,2] + 17.215;
   1:L PR[91] 10mm/sec CNT100;
   1:  PR[GP1:91,1] = PR[GP1:90,1] + 9.988;
   1:  PR[GP1:91,2] = PR[GP1:90,2] + 15.811;
   1:L PR[91] 10mm/sec CNT100;
   1:  PR[GP1:91,1] = PR[GP1:90,1] + 6.775;
   1:  PR[GP1:91,2] = PR[GP1:90,2] + 6.654;
   1:L PR[91] 10mm/sec CNT100;
   1:  PR[GP1:91,1] = PR[GP1:90,1] + 6.369;
   1:  PR[GP1:91,2] = PR[GP1:90,2] + 5.024;
   1:L PR[91] 10mm/sec CNT100;
   1:  PR[GP1:91,1] = PR[GP1:90,1] + 4.540;
   1:  PR[GP1:91,2] = PR[GP1:90,2] + 1.719;
   1:L PR[91] 10mm/sec CNT100;
   1:  PR[GP1:91,1] = PR[GP1:90,1] + 0.971;
   1:  PR[GP1:91,2] = PR[GP1:90,2] + 0.396;
   1:L PR[91] 10mm/sec CNT100;
   1:  PR[GP1:91,1] = PR[GP1:90,1] + -0.150;
   1:L PR[91] 10mm/sec CNT100;
   1:  PR[GP1:91,1] = PR[GP1:90,1] + -3.719;
   1:  PR[GP1:91,2] = PR[GP1:90,2] + 1.719;
   1:  PR[GP1:91,3] = PR[GP1:90,3] + 3.990;
   1:L PR[91] 10mm/sec CNT100;
   1:  PR[GP1:91,1] = PR[GP1:90,1] + -5.535;
   1:  PR[GP1:91,2] = PR[GP1:90,2] + 4.999;
   1:L PR[91] 10mm/sec CNT100;
   1:  PR[GP1:91,1] = PR[GP1:90,1] + -8.077;
   1:  PR[GP1:91,2] = PR[GP1:90,2] + 12.244;
   1:L PR[91] 10mm/sec CNT100;
   1:  PR[GP1:91,1] = PR[GP1:90,1] + -8.726;
   1:  PR[GP1:91,2] = PR[GP1:90,2] + 14.851;
   1:L PR[91] 10mm/sec CNT100;
   1:  PR[GP1:91,1] = PR[GP1:90,1] + -9.802;
   1:  PR[GP1:91,2] = PR[GP1:90,2] + 17.190;
   1:L PR[91] 10mm/sec CNT100;
   1:  PR[GP1:91,1] = PR[GP1:90,1] + -14.729;
   1:  PR[GP1:91,2] = PR[GP1:90,2] + 22.908;
   1:L PR[91] 10mm/sec CNT100;
   1:  PR[GP1:91,1] = PR[GP1:90,1] + -16.285;
   1:  PR[GP1:91,2] = PR[GP1:90,2] + 25.098;
   1:L PR[91] 10mm/sec CNT100;
   1:  PR[GP1:91,1] = PR[GP1:90,1] + -18.141;
   1:  PR[GP1:91,2] = PR[GP1:90,2] + 26.883;
   1:L PR[91] 10mm/sec CNT100;
   1:  PR[GP1:91,1] = PR[GP1:90,1] + -24.812;
   1:  PR[GP1:91,2] = PR[GP1:90,2] + 30.405;
   1:L PR[91] 10mm/sec CNT100;
   1:  PR[GP1:91,1] = PR[GP1:90,1] + -27.061;
   1:  PR[GP1:91,2] = PR[GP1:90,2] + 31.875;
   1:L PR[91] 10mm/sec CNT100;
   1:  PR[GP1:91,1] = PR[GP1:90,1] + -29.440;
   1:  PR[GP1:91,2] = PR[GP1:90,2] + 32.859;
   1:L PR[91] 10mm/sec CNT100;
   1:  PR[GP1:91,1] = PR[GP1:90,1] + -36.940;
   1:  PR[GP1:91,2] = PR[GP1:90,2] + 33.701;
   1:L PR[91] 10mm/sec CNT100;
   1:  PR[GP1:91,1] = PR[GP1:90,1] + -39.571;
   1:  PR[GP1:91,2] = PR[GP1:90,2] + 34.248;
   1:L PR[91] 10mm/sec CNT100;
   1:  PR[GP1:91,1] = PR[GP1:90,1] + -42.145;
   1:  PR[GP1:91,2] = PR[GP1:90,2] + 34.295;
   1:L PR[91] 10mm/sec CNT100;
   1:  PR[GP1:91,1] = PR[GP1:90,1] + -49.434;
   1:  PR[GP1:91,2] = PR[GP1:90,2] + 32.340;
   1:L PR[91] 10mm/sec CNT100;
   1:  PR[GP1:91,1] = PR[GP1:90,1] + -52.083;
   1:  PR[GP1:91,2] = PR[GP1:90,2] + 31.888;
   1:L PR[91] 10mm/sec CNT100;
   1:  PR[GP1:91,1] = PR[GP1:90,1] + -54.497;
   1:  PR[GP1:91,2] = PR[GP1:90,2] + 30.992;
   1:L PR[91] 10mm/sec CNT100;
   1:  PR[GP1:91,1] = PR[GP1:90,1] + -60.566;
   1:  PR[GP1:91,2] = PR[GP1:90,2] + 26.511;
   1:L PR[91] 10mm/sec CNT100;
   1:  PR[GP1:91,1] = PR[GP1:90,1] + -62.867;
   1:  PR[GP1:91,2] = PR[GP1:90,2] + 25.123;
   1:L PR[91] 10mm/sec CNT100;
   1:  PR[GP1:91,1] = PR[GP1:90,1] + -64.786;
   1:  PR[GP1:91,2] = PR[GP1:90,2] + 23.407;
   1:L PR[91] 10mm/sec CNT100;
   1:  PR[GP1:91,1] = PR[GP1:90,1] + -68.802;
   1:  PR[GP1:91,2] = PR[GP1:90,2] + 17.015;
   1:L PR[91] 10mm/sec CNT100;
   1:  PR[GP1:91,1] = PR[GP1:90,1] + -70.438;
   1:  PR[GP1:91,2] = PR[GP1:90,2] + 14.883;
   1:L PR[91] 10mm/sec CNT100;
   1:  PR[GP1:91,1] = PR[GP1:90,1] + -71.597;
   1:  PR[GP1:91,2] = PR[GP1:90,2] + 12.585;
   1:L PR[91] 10mm/sec CNT100;
   1:  PR[GP1:91,1] = PR[GP1:90,1] + -73.000;
   1:  PR[GP1:91,2] = PR[GP1:90,2] + 5.169;
   1:L PR[91] 10mm/sec CNT100;
   1:  PR[GP1:91,1] = PR[GP1:90,1] + -73.744;
   1:  PR[GP1:91,2] = PR[GP1:90,2] + 2.587;
   1:L PR[91] 10mm/sec CNT100;
   1:  PR[GP1:91,1] = PR[GP1:90,1] + -73.984;
   1:  PR[GP1:91,2] = PR[GP1:90,2] + 0.024;
   1:L PR[91] 10mm/sec CNT100;
   1:  PR[GP1:91,1] = PR[GP1:90,1] + -72.581;
   1:  PR[GP1:91,2] = PR[GP1:90,2] + -7.391;
   1:L PR[91] 10mm/sec CNT100;
   1:  PR[GP1:91,1] = PR[GP1:90,1] + -72.331;
   1:  PR[GP1:91,2] = PR[GP1:90,2] + -10.067;
   1:L PR[91] 10mm/sec CNT100;
   1:  PR[GP1:91,1] = PR[GP1:90,1] + -71.610;
   1:  PR[GP1:91,2] = PR[GP1:90,2] + -12.568;
   1:L PR[91] 10mm/sec CNT100;
   1:  PR[GP1:91,1] = PR[GP1:90,1] + -70.425;
   1:  PR[GP1:91,2] = PR[GP1:90,2] + -14.917;
   1:L PR[91] 10mm/sec CNT100;
   1:  PR[GP1:91,1] = PR[GP1:90,1] + -66.409;
   1:  PR[GP1:91,2] = PR[GP1:90,2] + -21.310;
   1:L PR[91] 10mm/sec CNT100;
   1:  PR[GP1:91,1] = PR[GP1:90,1] + -64.808;
   1:  PR[GP1:91,2] = PR[GP1:90,2] + -23.397;
   1:L PR[91] 10mm/sec CNT100;
   1:  PR[GP1:91,1] = PR[GP1:90,1] + -62.846;
   1:  PR[GP1:91,2] = PR[GP1:90,2] + -25.151;
   1:L PR[91] 10mm/sec CNT100;
   1:  PR[GP1:91,1] = PR[GP1:90,1] + -56.777;
   1:  PR[GP1:91,2] = PR[GP1:90,2] + -29.632;
   1:L PR[91] 10mm/sec CNT100;
   1:  PR[GP1:91,1] = PR[GP1:90,1] + -54.523;
   1:  PR[GP1:91,2] = PR[GP1:90,2] + -30.991;
   1:L PR[91] 10mm/sec CNT100;
   1:  PR[GP1:91,1] = PR[GP1:90,1] + -52.057;
   1:  PR[GP1:91,2] = PR[GP1:90,2] + -31.907;
   1:L PR[91] 10mm/sec CNT100;
   1:  PR[GP1:91,1] = PR[GP1:90,1] + -44.767;
   1:  PR[GP1:91,2] = PR[GP1:90,2] + -33.862;
   1:L PR[91] 10mm/sec CNT100;
   1:  PR[GP1:91,1] = PR[GP1:90,1] + -42.173;
   1:  PR[GP1:91,2] = PR[GP1:90,2] + -34.304;
   1:L PR[91] 10mm/sec CNT100;
   1:  PR[GP1:91,1] = PR[GP1:90,1] + -39.543;
   1:  PR[GP1:91,2] = PR[GP1:90,2] + -34.256;
   1:L PR[91] 10mm/sec CNT100;
   1:  PR[GP1:91,1] = PR[GP1:90,1] + -32.043;
   1:  PR[GP1:91,2] = PR[GP1:90,2] + -33.414;
   1:L PR[91] 10mm/sec CNT100;
   1:  PR[GP1:91,1] = PR[GP1:90,1] + -29.467;
   1:  PR[GP1:91,2] = PR[GP1:90,2] + -32.878;
   1:L PR[91] 10mm/sec CNT100;
   1:  PR[GP1:91,1] = PR[GP1:90,1] + -27.035;
   1:  PR[GP1:91,2] = PR[GP1:90,2] + -31.873;
   1:L PR[91] 10mm/sec CNT100;
   1:  PR[GP1:91,1] = PR[GP1:90,1] + -20.364;
   1:  PR[GP1:91,2] = PR[GP1:90,2] + -28.351;
   1:L PR[91] 10mm/sec CNT100;
   1:  PR[GP1:91,1] = PR[GP1:90,1] + -18.161;
   1:  PR[GP1:91,2] = PR[GP1:90,2] + -26.912;
   1:L PR[91] 10mm/sec CNT100;
   1:  PR[GP1:91,1] = PR[GP1:90,1] + -16.265;
   1:  PR[GP1:91,2] = PR[GP1:90,2] + -25.088;
   1:L PR[91] 10mm/sec CNT100;
   1:  PR[GP1:91,1] = PR[GP1:90,1] + -11.338;
   1:  PR[GP1:91,2] = PR[GP1:90,2] + -19.370;
   1:L PR[91] 10mm/sec CNT100;
   1:  PR[GP1:91,1] = PR[GP1:90,1] + -9.814;
   1:  PR[GP1:91,2] = PR[GP1:90,2] + -17.225;
   1:L PR[91] 10mm/sec CNT100;
   1:  PR[GP1:91,1] = PR[GP1:90,1] + -8.714;
   1:  PR[GP1:91,2] = PR[GP1:90,2] + -14.834;
   1:L PR[91] 10mm/sec CNT100;
   1:  PR[GP1:91,1] = PR[GP1:90,1] + -6.217;
   1:  PR[GP1:91,2] = PR[GP1:90,2] + -7.717;
   1:L PR[91] 10mm/sec CNT100;
   1:  PR[GP1:91,1] = PR[GP1:90,1] + -5.549;
   1:  PR[GP1:91,2] = PR[GP1:90,2] + -5.033;
   1:L PR[91] 10mm/sec CNT100;
   1:  PR[GP1:91,1] = PR[GP1:90,1] + -3.719;
   1:  PR[GP1:91,2] = PR[GP1:90,2] + -1.728;
   1:L PR[91] 10mm/sec CNT100;
   1:  PR[GP1:91,1] = PR[GP1:90,1] + -0.150;
   1:  PR[GP1:91,2] = PR[GP1:90,2] + -0.404;
   1:L PR[91] 10mm/sec CNT100;
   1:  PR[GP1:91,1] = PR[GP1:90,1] + 0.971;
   1:L PR[91] 10mm/sec CNT100;
   1:  PR[GP1:91,1] = PR[GP1:90,1] + 4.540;
   1:  PR[GP1:91,2] = PR[GP1:90,2] + -1.728;
   1:L PR[91] 10mm/sec CNT100;
   1:  PR[GP1:91,1] = PR[GP1:90,1] + 6.356;
   1:  PR[GP1:91,2] = PR[GP1:90,2] + -5.008;
   1:L PR[91] 10mm/sec CNT100;
   1:  PR[GP1:91,1] = PR[GP1:90,1] + 8.898;
   1:  PR[GP1:91,2] = PR[GP1:90,2] + -12.252;
   1:L PR[91] 10mm/sec CNT100;
   1:  PR[GP1:91,1] = PR[GP1:90,1] + 9.547;
   1:  PR[GP1:91,2] = PR[GP1:90,2] + -14.860;
   1:L PR[91] 10mm/sec CNT100;
   1:  PR[GP1:91,1] = PR[GP1:90,1] + 10.622;
   1:  PR[GP1:91,2] = PR[GP1:90,2] + -17.199;
   1:L PR[91] 10mm/sec CNT100;
   1:  PR[GP1:91,1] = PR[GP1:90,1] + 15.549;
   1:  PR[GP1:91,2] = PR[GP1:90,2] + -22.917;
   1:L PR[91] 10mm/sec CNT100;
   1:  PR[GP1:91,1] = PR[GP1:90,1] + 17.106;
   1:  PR[GP1:91,2] = PR[GP1:90,2] + -25.107;
   1:L PR[91] 10mm/sec CNT100;
   1:  PR[GP1:91,1] = PR[GP1:90,1] + 18.962;
   1:  PR[GP1:91,2] = PR[GP1:90,2] + -26.892;
   1:L PR[91] 10mm/sec CNT100;
   1:  PR[GP1:91,1] = PR[GP1:90,1] + 25.633;
   1:  PR[GP1:91,2] = PR[GP1:90,2] + -30.413;
   1:L PR[91] 10mm/sec CNT100;
   1:  PR[GP1:91,1] = PR[GP1:90,1] + 27.882;
   1:  PR[GP1:91,2] = PR[GP1:90,2] + -31.884;
   1:L PR[91] 10mm/sec CNT100;
   1:  PR[GP1:91,1] = PR[GP1:90,1] + 30.261;
   1:  PR[GP1:91,2] = PR[GP1:90,2] + -32.868;
   1:L PR[91] 10mm/sec CNT100;
   1:  PR[GP1:91,1] = PR[GP1:90,1] + 37.761;
   1:  PR[GP1:91,2] = PR[GP1:90,2] + -33.710;
   1:L PR[91] 10mm/sec CNT100;
   1:  PR[GP1:91,1] = PR[GP1:90,1] + 40.392;
   1:  PR[GP1:91,2] = PR[GP1:90,2] + -34.257;
   1:L PR[91] 10mm/sec CNT100;
   1:  PR[GP1:91,1] = PR[GP1:90,1] + 42.966;
   1:  PR[GP1:91,2] = PR[GP1:90,2] + -34.304;
   1:L PR[91] 10mm/sec CNT100;
   1:  PR[GP1:91,1] = PR[GP1:90,1] + 50.255;
   1:  PR[GP1:91,2] = PR[GP1:90,2] + -32.349;
   1:L PR[91] 10mm/sec CNT100;
   1:  PR[GP1:91,1] = PR[GP1:90,1] + 52.904;
   1:  PR[GP1:91,2] = PR[GP1:90,2] + -31.897;
   1:L PR[91] 10mm/sec CNT100;
   1:  PR[GP1:91,1] = PR[GP1:90,1] + 55.317;
   1:  PR[GP1:91,2] = PR[GP1:90,2] + -31.001;
   1:L PR[91] 10mm/sec CNT100;
   1:  PR[GP1:91,1] = PR[GP1:90,1] + 61.387;
   1:  PR[GP1:91,2] = PR[GP1:90,2] + -26.520;
   1:L PR[91] 10mm/sec CNT100;
   1:  PR[GP1:91,1] = PR[GP1:90,1] + 63.688;
   1:  PR[GP1:91,2] = PR[GP1:90,2] + -25.132;
   1:L PR[91] 10mm/sec CNT100;
   1:  PR[GP1:91,1] = PR[GP1:90,1] + 65.607;
   1:  PR[GP1:91,2] = PR[GP1:90,2] + -23.416;
   1:L PR[91] 10mm/sec CNT100;
   1:  PR[GP1:91,1] = PR[GP1:90,1] + 69.623;
   1:  PR[GP1:91,2] = PR[GP1:90,2] + -17.024;
   1:L PR[91] 10mm/sec CNT100;
   1:  PR[GP1:91,1] = PR[GP1:90,1] + 71.258;
   1:  PR[GP1:91,2] = PR[GP1:90,2] + -14.892;
   1:L PR[91] 10mm/sec CNT100;
   1:  PR[GP1:91,1] = PR[GP1:90,1] + 72.418;
   1:  PR[GP1:91,2] = PR[GP1:90,2] + -12.593;
   1:L PR[91] 10mm/sec CNT100;
   1:  PR[GP1:91,1] = PR[GP1:90,1] + 73.821;
   1:  PR[GP1:91,2] = PR[GP1:90,2] + -5.178;
   1:L PR[91] 10mm/sec CNT100;
   1:  PR[GP1:91,1] = PR[GP1:90,1] + 74.565;
   1:  PR[GP1:91,2] = PR[GP1:90,2] + -2.596;
   1:L PR[91] 10mm/sec CNT100;
   1:  PR[GP1:91,1] = PR[GP1:90,1] + 74.805;
   1:  PR[GP1:91,2] = PR[GP1:90,2] + -0.033;
   1:L PR[91] 10mm/sec CNT100;
   1:  PR[GP1:91,1] = PR[GP1:90,1] + 73.402;
   1:  PR[GP1:91,2] = PR[GP1:90,2] + 7.382;
   1:L PR[91] 10mm/sec CNT100;
   1:  PR[GP1:91,1] = PR[GP1:90,1] + 73.151;
   1:  PR[GP1:91,2] = PR[GP1:90,2] + 10.058;
   1:L PR[91] 10mm/sec CNT100;
   1:  PR[GP1:91,1] = PR[GP1:90,1] + 72.431;
   1:  PR[GP1:91,2] = PR[GP1:90,2] + 12.559;
   1:L PR[91] 10mm/sec CNT100;
   1:  PR[GP1:91,1] = PR[GP1:90,1] + 71.246;
   1:  PR[GP1:91,2] = PR[GP1:90,2] + 14.908;
   1:L PR[91] 10mm/sec CNT100;
   1:  PR[GP1:91,1] = PR[GP1:90,1] + 67.229;
   1:  PR[GP1:91,2] = PR[GP1:90,2] + 21.301;
   1:L PR[91] 10mm/sec CNT100;
   1:  PR[GP1:91,1] = PR[GP1:90,1] + 65.628;
   1:  PR[GP1:91,2] = PR[GP1:90,2] + 23.388;
   1:L PR[91] 10mm/sec CNT100;
   1:  PR[GP1:91,1] = PR[GP1:90,1] + 63.667;
   1:  PR[GP1:91,2] = PR[GP1:90,2] + 25.142;
   1:L PR[91] 10mm/sec CNT100;
   1:  PR[GP1:91,1] = PR[GP1:90,1] + 57.597;
   1:  PR[GP1:91,2] = PR[GP1:90,2] + 29.623;
   1:L PR[91] 10mm/sec CNT100;
   1:  PR[GP1:91,1] = PR[GP1:90,1] + 55.344;
   1:  PR[GP1:91,2] = PR[GP1:90,2] + 30.982;
   1:L PR[91] 10mm/sec CNT100;
   1:  PR[GP1:91,1] = PR[GP1:90,1] + 52.878;
   1:  PR[GP1:91,2] = PR[GP1:90,2] + 31.898;
   1:L PR[91] 10mm/sec CNT100;
   1:  PR[GP1:91,1] = PR[GP1:90,1] + 45.588;
   1:  PR[GP1:91,2] = PR[GP1:90,2] + 33.854;
   1:L PR[91] 10mm/sec CNT100;
   1:  PR[GP1:91,1] = PR[GP1:90,1] + 42.994;
   1:  PR[GP1:91,2] = PR[GP1:90,2] + 34.295;
   1:L PR[91] 10mm/sec CNT100;
   1:  PR[GP1:91,1] = PR[GP1:90,1] + 40.363;
   1:  PR[GP1:91,2] = PR[GP1:90,2] + 34.248;
   1:L PR[91] 10mm/sec CNT100;
   1:  PR[GP1:91,1] = PR[GP1:90,1] + 32.863;
   1:  PR[GP1:91,2] = PR[GP1:90,2] + 33.405;
   1:L PR[91] 10mm/sec CNT100;
   1:  PR[GP1:91,1] = PR[GP1:90,1] + 30.287;
   1:  PR[GP1:91,2] = PR[GP1:90,2] + 32.870;
   1:L PR[91] 10mm/sec CNT100;
   1:  PR[GP1:91,1] = PR[GP1:90,1] + 27.856;
   1:  PR[GP1:91,2] = PR[GP1:90,2] + 31.864;
   1:L PR[91] 10mm/sec CNT100;
   1:  PR[GP1:91,1] = PR[GP1:90,1] + 21.184;
   1:  PR[GP1:91,2] = PR[GP1:90,2] + 28.343;
   1:L PR[91] 10mm/sec CNT100;
   1:  PR[GP1:91,1] = PR[GP1:90,1] + 18.982;
   1:  PR[GP1:91,2] = PR[GP1:90,2] + 26.903;
   1:L PR[91] 10mm/sec CNT100;
   1:  PR[GP1:91,1] = PR[GP1:90,1] + 17.086;
   1:  PR[GP1:91,2] = PR[GP1:90,2] + 25.079;
   1:L PR[91] 10mm/sec CNT100;
   1:  PR[GP1:91,1] = PR[GP1:90,1] + 12.159;
   1:  PR[GP1:91,2] = PR[GP1:90,2] + 19.361;
   1:L PR[91] 10mm/sec CNT100;
   1:  PR[GP1:91,1] = PR[GP1:90,1] + 10.634;
   1:  PR[GP1:91,2] = PR[GP1:90,2] + 17.216;
   1:L PR[91] 10mm/sec CNT100;
   1:  PR[GP1:91,1] = PR[GP1:90,1] + 9.535;
   1:  PR[GP1:91,2] = PR[GP1:90,2] + 14.826;
   1:L PR[91] 10mm/sec CNT100;
   1:  PR[GP1:91,1] = PR[GP1:90,1] + 7.038;
   1:  PR[GP1:91,2] = PR[GP1:90,2] + 7.708;
   1:L PR[91] 10mm/sec CNT100;
   1:  PR[GP1:91,1] = PR[GP1:90,1] + 6.369;
   1:  PR[GP1:91,2] = PR[GP1:90,2] + 5.024;
   1:L PR[91] 10mm/sec CNT100;
   1:  PR[GP1:91,1] = PR[GP1:90,1] + 4.540;
   1:  PR[GP1:91,2] = PR[GP1:90,2] + 1.719;
   1:L PR[91] 10mm/sec CNT100;
   1:  PR[GP1:91,1] = PR[GP1:90,1] + 0.971;
   1:  PR[GP1:91,2] = PR[GP1:90,2] + 0.396;
   1:L PR[91] 10mm/sec CNT100;
   1:  PR[GP1:91,1] = PR[GP1:90,1] + -0.150;
   1:L PR[91] 10mm/sec CNT100;
   1:  PR[GP1:91,1] = PR[GP1:90,1] + -3.719;
   1:  PR[GP1:91,2] = PR[GP1:90,2] + 1.719;
   1:  PR[GP1:91,3] = PR[GP1:90,3] + 5.320;
   1:L PR[91] 10mm/sec CNT100;
   1:  PR[GP1:91,1] = PR[GP1:90,1] + -5.535;
   1:  PR[GP1:91,2] = PR[GP1:90,2] + 4.999;
   1:L PR[91] 10mm/sec CNT100;
   1:  PR[GP1:91,1] = PR[GP1:90,1] + -7.361;
   1:  PR[GP1:91,2] = PR[GP1:90,2] + 10.204;
   1:L PR[91] 10mm/sec CNT100;
   1:  PR[GP1:91,1] = PR[GP1:90,1] + -8.273;
   1:  PR[GP1:91,2] = PR[GP1:90,2] + 13.865;
   1:L PR[91] 10mm/sec CNT100;
   1:  PR[GP1:91,1] = PR[GP1:90,1] + -9.802;
   1:  PR[GP1:91,2] = PR[GP1:90,2] + 17.191;
   1:L PR[91] 10mm/sec CNT100;
   1:  PR[GP1:91,1] = PR[GP1:90,1] + -13.317;
   1:  PR[GP1:91,2] = PR[GP1:90,2] + 21.270;
   1:L PR[91] 10mm/sec CNT100;
   1:  PR[GP1:91,1] = PR[GP1:90,1] + -15.503;
   1:  PR[GP1:91,2] = PR[GP1:90,2] + 24.346;
   1:L PR[91] 10mm/sec CNT100;
   1:  PR[GP1:91,1] = PR[GP1:90,1] + -18.141;
   1:  PR[GP1:91,2] = PR[GP1:90,2] + 26.883;
   1:L PR[91] 10mm/sec CNT100;
   1:  PR[GP1:91,1] = PR[GP1:90,1] + -22.900;
   1:  PR[GP1:91,2] = PR[GP1:90,2] + 29.396;
   1:L PR[91] 10mm/sec CNT100;
   1:  PR[GP1:91,1] = PR[GP1:90,1] + -26.059;
   1:  PR[GP1:91,2] = PR[GP1:90,2] + 31.460;
   1:L PR[91] 10mm/sec CNT100;
   1:  PR[GP1:91,1] = PR[GP1:90,1] + -29.442;
   1:  PR[GP1:91,2] = PR[GP1:90,2] + 32.859;
   1:L PR[91] 10mm/sec CNT100;
   1:  PR[GP1:91,1] = PR[GP1:90,1] + -34.792;
   1:  PR[GP1:91,2] = PR[GP1:90,2] + 33.460;
   1:L PR[91] 10mm/sec CNT100;
   1:  PR[GP1:91,1] = PR[GP1:90,1] + -38.486;
   1:  PR[GP1:91,2] = PR[GP1:90,2] + 34.228;
   1:L PR[91] 10mm/sec CNT100;
   1:  PR[GP1:91,1] = PR[GP1:90,1] + -42.146;
   1:  PR[GP1:91,2] = PR[GP1:90,2] + 34.295;
   1:L PR[91] 10mm/sec CNT100;
   1:  PR[GP1:91,1] = PR[GP1:90,1] + -47.346;
   1:  PR[GP1:91,2] = PR[GP1:90,2] + 32.900;
   1:L PR[91] 10mm/sec CNT100;
   1:  PR[GP1:91,1] = PR[GP1:90,1] + -51.066;
   1:  PR[GP1:91,2] = PR[GP1:90,2] + 32.266;
   1:L PR[91] 10mm/sec CNT100;
   1:  PR[GP1:91,1] = PR[GP1:90,1] + -54.497;
   1:  PR[GP1:91,2] = PR[GP1:90,2] + 30.992;
   1:L PR[91] 10mm/sec CNT100;
   1:  PR[GP1:91,1] = PR[GP1:90,1] + -58.827;
   1:  PR[GP1:91,2] = PR[GP1:90,2] + 27.795;
   1:L PR[91] 10mm/sec CNT100;
   1:  PR[GP1:91,1] = PR[GP1:90,1] + -62.058;
   1:  PR[GP1:91,2] = PR[GP1:90,2] + 25.847;
   1:L PR[91] 10mm/sec CNT100;
   1:  PR[GP1:91,1] = PR[GP1:90,1] + -64.787;
   1:  PR[GP1:91,2] = PR[GP1:90,2] + 23.407;
   1:L PR[91] 10mm/sec CNT100;
   1:  PR[GP1:91,1] = PR[GP1:90,1] + -67.652;
   1:  PR[GP1:91,2] = PR[GP1:90,2] + 18.847;
   1:L PR[91] 10mm/sec CNT100;
   1:  PR[GP1:91,1] = PR[GP1:90,1] + -69.948;
   1:  PR[GP1:91,2] = PR[GP1:90,2] + 15.853;
   1:L PR[91] 10mm/sec CNT100;
   1:  PR[GP1:91,1] = PR[GP1:90,1] + -71.598;
   1:  PR[GP1:91,2] = PR[GP1:90,2] + 12.584;
   1:L PR[91] 10mm/sec CNT100;
   1:  PR[GP1:91,1] = PR[GP1:90,1] + -72.598;
   1:  PR[GP1:91,2] = PR[GP1:90,2] + 7.295;
   1:L PR[91] 10mm/sec CNT100;
   1:  PR[GP1:91,1] = PR[GP1:90,1] + -73.643;
   1:  PR[GP1:91,2] = PR[GP1:90,2] + 3.669;
   1:L PR[91] 10mm/sec CNT100;
   1:  PR[GP1:91,1] = PR[GP1:90,1] + -73.984;
   1:  PR[GP1:91,2] = PR[GP1:90,2] + 0.024;
   1:L PR[91] 10mm/sec CNT100;
   1:  PR[GP1:91,1] = PR[GP1:90,1] + -72.984;
   1:  PR[GP1:91,2] = PR[GP1:90,2] + -5.266;
   1:L PR[91] 10mm/sec CNT100;
   1:  PR[GP1:91,1] = PR[GP1:90,1] + -72.631;
   1:  PR[GP1:91,2] = PR[GP1:90,2] + -9.023;
   1:L PR[91] 10mm/sec CNT100;
   1:  PR[GP1:91,1] = PR[GP1:90,1] + -71.610;
   1:  PR[GP1:91,2] = PR[GP1:90,2] + -12.568;
   1:L PR[91] 10mm/sec CNT100;
   1:  PR[GP1:91,1] = PR[GP1:90,1] + -69.936;
   1:  PR[GP1:91,2] = PR[GP1:90,2] + -15.886;
   1:L PR[91] 10mm/sec CNT100;
   1:  PR[GP1:91,1] = PR[GP1:90,1] + -67.071;
   1:  PR[GP1:91,2] = PR[GP1:90,2] + -20.447;
   1:L PR[91] 10mm/sec CNT100;
   1:  PR[GP1:91,1] = PR[GP1:90,1] + -64.808;
   1:  PR[GP1:91,2] = PR[GP1:90,2] + -23.396;
   1:L PR[91] 10mm/sec CNT100;
   1:  PR[GP1:91,1] = PR[GP1:90,1] + -62.037;
   1:  PR[GP1:91,2] = PR[GP1:90,2] + -25.874;
   1:L PR[91] 10mm/sec CNT100;
   1:  PR[GP1:91,1] = PR[GP1:90,1] + -57.707;
   1:  PR[GP1:91,2] = PR[GP1:90,2] + -29.071;
   1:L PR[91] 10mm/sec CNT100;
   1:  PR[GP1:91,1] = PR[GP1:90,1] + -54.524;
   1:  PR[GP1:91,2] = PR[GP1:90,2] + -30.991;
   1:L PR[91] 10mm/sec CNT100;
   1:  PR[GP1:91,1] = PR[GP1:90,1] + -51.039;
   1:  PR[GP1:91,2] = PR[GP1:90,2] + -32.285;
   1:L PR[91] 10mm/sec CNT100;
   1:  PR[GP1:91,1] = PR[GP1:90,1] + -45.839;
   1:  PR[GP1:91,2] = PR[GP1:90,2] + -33.680;
   1:L PR[91] 10mm/sec CNT100;
   1:  PR[GP1:91,1] = PR[GP1:90,1] + -42.174;
   1:  PR[GP1:91,2] = PR[GP1:90,2] + -34.304;
   1:L PR[91] 10mm/sec CNT100;
   1:  PR[GP1:91,1] = PR[GP1:90,1] + -38.458;
   1:  PR[GP1:91,2] = PR[GP1:90,2] + -34.237;
   1:L PR[91] 10mm/sec CNT100;
   1:  PR[GP1:91,1] = PR[GP1:90,1] + -33.107;
   1:  PR[GP1:91,2] = PR[GP1:90,2] + -33.636;
   1:L PR[91] 10mm/sec CNT100;
   1:  PR[GP1:91,1] = PR[GP1:90,1] + -29.468;
   1:  PR[GP1:91,2] = PR[GP1:90,2] + -32.879;
   1:L PR[91] 10mm/sec CNT100;
   1:  PR[GP1:91,1] = PR[GP1:90,1] + -26.033;
   1:  PR[GP1:91,2] = PR[GP1:90,2] + -31.458;
   1:L PR[91] 10mm/sec CNT100;
   1:  PR[GP1:91,1] = PR[GP1:90,1] + -21.273;
   1:  PR[GP1:91,2] = PR[GP1:90,2] + -28.946;
   1:L PR[91] 10mm/sec CNT100;
   1:  PR[GP1:91,1] = PR[GP1:90,1] + -18.162;
   1:  PR[GP1:91,2] = PR[GP1:90,2] + -26.912;
   1:L PR[91] 10mm/sec CNT100;
   1:  PR[GP1:91,1] = PR[GP1:90,1] + -15.483;
   1:  PR[GP1:91,2] = PR[GP1:90,2] + -24.335;
   1:L PR[91] 10mm/sec CNT100;
   1:  PR[GP1:91,1] = PR[GP1:90,1] + -11.968;
   1:  PR[GP1:91,2] = PR[GP1:90,2] + -20.256;
   1:L PR[91] 10mm/sec CNT100;
   1:  PR[GP1:91,1] = PR[GP1:90,1] + -9.814;
   1:  PR[GP1:91,2] = PR[GP1:90,2] + -17.226;
   1:L PR[91] 10mm/sec CNT100;
   1:  PR[GP1:91,1] = PR[GP1:90,1] + -8.261;
   1:  PR[GP1:91,2] = PR[GP1:90,2] + -13.848;
   1:L PR[91] 10mm/sec CNT100;
   1:  PR[GP1:91,1] = PR[GP1:90,1] + -6.480;
   1:  PR[GP1:91,2] = PR[GP1:90,2] + -8.771;
   1:L PR[91] 10mm/sec CNT100;
   1:  PR[GP1:91,1] = PR[GP1:90,1] + -5.549;
   1:  PR[GP1:91,2] = PR[GP1:90,2] + -5.033;
   1:L PR[91] 10mm/sec CNT100;
   1:  PR[GP1:91,1] = PR[GP1:90,1] + -3.719;
   1:  PR[GP1:91,2] = PR[GP1:90,2] + -1.728;
   1:L PR[91] 10mm/sec CNT100;
   1:  PR[GP1:91,1] = PR[GP1:90,1] + -0.150;
   1:  PR[GP1:91,2] = PR[GP1:90,2] + -0.404;
   1:L PR[91] 10mm/sec CNT100;
   1:  PR[GP1:91,1] = PR[GP1:90,1] + 0.971;
   1:L PR[91] 10mm/sec CNT100;
   1:  PR[GP1:91,1] = PR[GP1:90,1] + 4.540;
   1:  PR[GP1:91,2] = PR[GP1:90,2] + -1.728;
   1:L PR[91] 10mm/sec CNT100;
   1:  PR[GP1:91,1] = PR[GP1:90,1] + 6.356;
   1:  PR[GP1:91,2] = PR[GP1:90,2] + -5.008;
   1:L PR[91] 10mm/sec CNT100;
   1:  PR[GP1:91,1] = PR[GP1:90,1] + 8.182;
   1:  PR[GP1:91,2] = PR[GP1:90,2] + -10.213;
   1:L PR[91] 10mm/sec CNT100;
   1:  PR[GP1:91,1] = PR[GP1:90,1] + 9.094;
   1:  PR[GP1:91,2] = PR[GP1:90,2] + -13.874;
   1:L PR[91] 10mm/sec CNT100;
   1:  PR[GP1:91,1] = PR[GP1:90,1] + 10.623;
   1:  PR[GP1:91,2] = PR[GP1:90,2] + -17.200;
   1:L PR[91] 10mm/sec CNT100;
   1:  PR[GP1:91,1] = PR[GP1:90,1] + 14.138;
   1:  PR[GP1:91,2] = PR[GP1:90,2] + -21.279;
   1:L PR[91] 10mm/sec CNT100;
   1:  PR[GP1:91,1] = PR[GP1:90,1] + 16.324;
   1:  PR[GP1:91,2] = PR[GP1:90,2] + -24.355;
   1:L PR[91] 10mm/sec CNT100;
   1:  PR[GP1:91,1] = PR[GP1:90,1] + 18.962;
   1:  PR[GP1:91,2] = PR[GP1:90,2] + -26.892;
   1:L PR[91] 10mm/sec CNT100;
   1:  PR[GP1:91,1] = PR[GP1:90,1] + 23.721;
   1:  PR[GP1:91,2] = PR[GP1:90,2] + -29.404;
   1:L PR[91] 10mm/sec CNT100;
   1:  PR[GP1:91,1] = PR[GP1:90,1] + 26.879;
   1:  PR[GP1:91,2] = PR[GP1:90,2] + -31.469;
   1:L PR[91] 10mm/sec CNT100;
   1:  PR[GP1:91,1] = PR[GP1:90,1] + 30.262;
   1:  PR[GP1:91,2] = PR[GP1:90,2] + -32.868;
   1:L PR[91] 10mm/sec CNT100;
   1:  PR[GP1:91,1] = PR[GP1:90,1] + 35.612;
   1:  PR[GP1:91,2] = PR[GP1:90,2] + -33.469;
   1:L PR[91] 10mm/sec CNT100;
   1:  PR[GP1:91,1] = PR[GP1:90,1] + 39.306;
   1:  PR[GP1:91,2] = PR[GP1:90,2] + -34.237;
   1:L PR[91] 10mm/sec CNT100;
   1:  PR[GP1:91,1] = PR[GP1:90,1] + 42.967;
   1:  PR[GP1:91,2] = PR[GP1:90,2] + -34.304;
   1:L PR[91] 10mm/sec CNT100;
   1:  PR[GP1:91,1] = PR[GP1:90,1] + 48.167;
   1:  PR[GP1:91,2] = PR[GP1:90,2] + -32.909;
   1:L PR[91] 10mm/sec CNT100;
   1:  PR[GP1:91,1] = PR[GP1:90,1] + 51.886;
   1:  PR[GP1:91,2] = PR[GP1:90,2] + -32.275;
   1:L PR[91] 10mm/sec CNT100;
   1:  PR[GP1:91,1] = PR[GP1:90,1] + 55.318;
   1:  PR[GP1:91,2] = PR[GP1:90,2] + -31.000;
   1:L PR[91] 10mm/sec CNT100;
   1:  PR[GP1:91,1] = PR[GP1:90,1] + 59.648;
   1:  PR[GP1:91,2] = PR[GP1:90,2] + -27.804;
   1:L PR[91] 10mm/sec CNT100;
   1:  PR[GP1:91,1] = PR[GP1:90,1] + 62.879;
   1:  PR[GP1:91,2] = PR[GP1:90,2] + -25.855;
   1:L PR[91] 10mm/sec CNT100;
   1:  PR[GP1:91,1] = PR[GP1:90,1] + 65.608;
   1:  PR[GP1:91,2] = PR[GP1:90,2] + -23.415;
   1:L PR[91] 10mm/sec CNT100;
   1:  PR[GP1:91,1] = PR[GP1:90,1] + 68.473;
   1:  PR[GP1:91,2] = PR[GP1:90,2] + -18.855;
   1:L PR[91] 10mm/sec CNT100;
   1:  PR[GP1:91,1] = PR[GP1:90,1] + 70.769;
   1:  PR[GP1:91,2] = PR[GP1:90,2] + -15.861;
   1:L PR[91] 10mm/sec CNT100;
   1:  PR[GP1:91,1] = PR[GP1:90,1] + 72.418;
   1:  PR[GP1:91,2] = PR[GP1:90,2] + -12.593;
   1:L PR[91] 10mm/sec CNT100;
   1:  PR[GP1:91,1] = PR[GP1:90,1] + 73.419;
   1:  PR[GP1:91,2] = PR[GP1:90,2] + -7.303;
   1:L PR[91] 10mm/sec CNT100;
   1:  PR[GP1:91,1] = PR[GP1:90,1] + 74.463;
   1:  PR[GP1:91,2] = PR[GP1:90,2] + -3.677;
   1:L PR[91] 10mm/sec CNT100;
   1:  PR[GP1:91,1] = PR[GP1:90,1] + 74.805;
   1:  PR[GP1:91,2] = PR[GP1:90,2] + -0.033;
   1:L PR[91] 10mm/sec CNT100;
   1:  PR[GP1:91,1] = PR[GP1:90,1] + 73.804;
   1:  PR[GP1:91,2] = PR[GP1:90,2] + 5.257;
   1:L PR[91] 10mm/sec CNT100;
   1:  PR[GP1:91,1] = PR[GP1:90,1] + 73.452;
   1:  PR[GP1:91,2] = PR[GP1:90,2] + 9.014;
   1:L PR[91] 10mm/sec CNT100;
   1:  PR[GP1:91,1] = PR[GP1:90,1] + 72.431;
   1:  PR[GP1:91,2] = PR[GP1:90,2] + 12.559;
   1:L PR[91] 10mm/sec CNT100;
   1:  PR[GP1:91,1] = PR[GP1:90,1] + 70.756;
   1:  PR[GP1:91,2] = PR[GP1:90,2] + 15.878;
   1:L PR[91] 10mm/sec CNT100;
   1:  PR[GP1:91,1] = PR[GP1:90,1] + 67.891;
   1:  PR[GP1:91,2] = PR[GP1:90,2] + 20.438;
   1:L PR[91] 10mm/sec CNT100;
   1:  PR[GP1:91,1] = PR[GP1:90,1] + 65.629;
   1:  PR[GP1:91,2] = PR[GP1:90,2] + 23.388;
   1:L PR[91] 10mm/sec CNT100;
   1:  PR[GP1:91,1] = PR[GP1:90,1] + 62.858;
   1:  PR[GP1:91,2] = PR[GP1:90,2] + 25.865;
   1:L PR[91] 10mm/sec CNT100;
   1:  PR[GP1:91,1] = PR[GP1:90,1] + 58.528;
   1:  PR[GP1:91,2] = PR[GP1:90,2] + 29.062;
   1:L PR[91] 10mm/sec CNT100;
   1:  PR[GP1:91,1] = PR[GP1:90,1] + 55.345;
   1:  PR[GP1:91,2] = PR[GP1:90,2] + 30.982;
   1:L PR[91] 10mm/sec CNT100;
   1:  PR[GP1:91,1] = PR[GP1:90,1] + 51.860;
   1:  PR[GP1:91,2] = PR[GP1:90,2] + 32.276;
   1:L PR[91] 10mm/sec CNT100;
   1:  PR[GP1:91,1] = PR[GP1:90,1] + 46.660;
   1:  PR[GP1:91,2] = PR[GP1:90,2] + 33.671;
   1:L PR[91] 10mm/sec CNT100;
   1:  PR[GP1:91,1] = PR[GP1:90,1] + 42.995;
   1:  PR[GP1:91,2] = PR[GP1:90,2] + 34.295;
   1:L PR[91] 10mm/sec CNT100;
   1:  PR[GP1:91,1] = PR[GP1:90,1] + 39.278;
   1:  PR[GP1:91,2] = PR[GP1:90,2] + 34.228;
   1:L PR[91] 10mm/sec CNT100;
   1:  PR[GP1:91,1] = PR[GP1:90,1] + 33.928;
   1:  PR[GP1:91,2] = PR[GP1:90,2] + 33.627;
   1:L PR[91] 10mm/sec CNT100;
   1:  PR[GP1:91,1] = PR[GP1:90,1] + 30.288;
   1:  PR[GP1:91,2] = PR[GP1:90,2] + 32.870;
   1:L PR[91] 10mm/sec CNT100;
   1:  PR[GP1:91,1] = PR[GP1:90,1] + 26.853;
   1:  PR[GP1:91,2] = PR[GP1:90,2] + 31.450;
   1:L PR[91] 10mm/sec CNT100;
   1:  PR[GP1:91,1] = PR[GP1:90,1] + 22.094;
   1:  PR[GP1:91,2] = PR[GP1:90,2] + 28.937;
   1:L PR[91] 10mm/sec CNT100;
   1:  PR[GP1:91,1] = PR[GP1:90,1] + 18.982;
   1:  PR[GP1:91,2] = PR[GP1:90,2] + 26.903;
   1:L PR[91] 10mm/sec CNT100;
   1:  PR[GP1:91,1] = PR[GP1:90,1] + 16.303;
   1:  PR[GP1:91,2] = PR[GP1:90,2] + 24.326;
   1:L PR[91] 10mm/sec CNT100;
   1:  PR[GP1:91,1] = PR[GP1:90,1] + 12.788;
   1:  PR[GP1:91,2] = PR[GP1:90,2] + 20.247;
   1:L PR[91] 10mm/sec CNT100;
   1:  PR[GP1:91,1] = PR[GP1:90,1] + 10.635;
   1:  PR[GP1:91,2] = PR[GP1:90,2] + 17.217;
   1:L PR[91] 10mm/sec CNT100;
   1:  PR[GP1:91,1] = PR[GP1:90,1] + 9.082;
   1:  PR[GP1:91,2] = PR[GP1:90,2] + 13.840;
   1:L PR[91] 10mm/sec CNT100;
   1:  PR[GP1:91,1] = PR[GP1:90,1] + 7.300;
   1:  PR[GP1:91,2] = PR[GP1:90,2] + 8.762;
   1:L PR[91] 10mm/sec CNT100;
   1:  PR[GP1:91,1] = PR[GP1:90,1] + 6.369;
   1:  PR[GP1:91,2] = PR[GP1:90,2] + 5.024;
   1:L PR[91] 10mm/sec CNT100;
   1:  PR[GP1:91,1] = PR[GP1:90,1] + 4.540;
   1:  PR[GP1:91,2] = PR[GP1:90,2] + 1.719;
   1:L PR[91] 10mm/sec CNT100;
   1:  PR[GP1:91,1] = PR[GP1:90,1] + 0.971;
   1:  PR[GP1:91,2] = PR[GP1:90,2] + 0.396;
   1:L PR[91] 10mm/sec CNT100;
   1:  PR[GP1:91,1] = PR[GP1:90,1] + -0.150;
   1:L PR[91] 10mm/sec CNT100;
   1:  PR[GP1:91,1] = PR[GP1:90,1] + -3.719;
   1:  PR[GP1:91,2] = PR[GP1:90,2] + 1.719;
   1:  PR[GP1:91,3] = PR[GP1:90,3] + 6.650;
   1:L PR[91] 10mm/sec CNT100;
   1:  PR[GP1:91,1] = PR[GP1:90,1] + -5.535;
   1:  PR[GP1:91,2] = PR[GP1:90,2] + 4.999;
   1:L PR[91] 10mm/sec CNT100;
   1:  PR[GP1:91,1] = PR[GP1:90,1] + -6.645;
   1:  PR[GP1:91,2] = PR[GP1:90,2] + 8.164;
   1:L PR[91] 10mm/sec CNT100;
   1:  PR[GP1:91,1] = PR[GP1:90,1] + -7.820;
   1:  PR[GP1:91,2] = PR[GP1:90,2] + 12.879;
   1:L PR[91] 10mm/sec CNT100;
   1:  PR[GP1:91,1] = PR[GP1:90,1] + -9.803;
   1:  PR[GP1:91,2] = PR[GP1:90,2] + 17.192;
   1:L PR[91] 10mm/sec CNT100;
   1:  PR[GP1:91,1] = PR[GP1:90,1] + -11.905;
   1:  PR[GP1:91,2] = PR[GP1:90,2] + 19.632;
   1:L PR[91] 10mm/sec CNT100;
   1:  PR[GP1:91,1] = PR[GP1:90,1] + -14.721;
   1:  PR[GP1:91,2] = PR[GP1:90,2] + 23.593;
   1:L PR[91] 10mm/sec CNT100;
   1:  PR[GP1:91,1] = PR[GP1:90,1] + -18.142;
   1:  PR[GP1:91,2] = PR[GP1:90,2] + 26.884;
   1:L PR[91] 10mm/sec CNT100;
   1:  PR[GP1:91,1] = PR[GP1:90,1] + -20.989;
   1:  PR[GP1:91,2] = PR[GP1:90,2] + 28.387;
   1:L PR[91] 10mm/sec CNT100;
   1:  PR[GP1:91,1] = PR[GP1:90,1] + -25.056;
   1:  PR[GP1:91,2] = PR[GP1:90,2] + 31.046;
   1:L PR[91] 10mm/sec CNT100;
   1:  PR[GP1:91,1] = PR[GP1:90,1] + -29.443;
   1:  PR[GP1:91,2] = PR[GP1:90,2] + 32.859;
   1:L PR[91] 10mm/sec CNT100;
   1:  PR[GP1:91,1] = PR[GP1:90,1] + -32.643;
   1:  PR[GP1:91,2] = PR[GP1:90,2] + 33.219;
   1:L PR[91] 10mm/sec CNT100;
   1:  PR[GP1:91,1] = PR[GP1:90,1] + -37.401;
   1:  PR[GP1:91,2] = PR[GP1:90,2] + 34.209;
   1:L PR[91] 10mm/sec CNT100;
   1:  PR[GP1:91,1] = PR[GP1:90,1] + -42.147;
   1:  PR[GP1:91,2] = PR[GP1:90,2] + 34.295;
   1:L PR[91] 10mm/sec CNT100;
   1:  PR[GP1:91,1] = PR[GP1:90,1] + -45.258;
   1:  PR[GP1:91,2] = PR[GP1:90,2] + 33.461;
   1:L PR[91] 10mm/sec CNT100;
   1:  PR[GP1:91,1] = PR[GP1:90,1] + -50.048;
   1:  PR[GP1:91,2] = PR[GP1:90,2] + 32.644;
   1:L PR[91] 10mm/sec CNT100;
   1:  PR[GP1:91,1] = PR[GP1:90,1] + -54.498;
   1:  PR[GP1:91,2] = PR[GP1:90,2] + 30.991;
   1:L PR[91] 10mm/sec CNT100;
   1:  PR[GP1:91,1] = PR[GP1:90,1] + -57.088;
   1:  PR[GP1:91,2] = PR[GP1:90,2] + 29.079;
   1:L PR[91] 10mm/sec CNT100;
   1:  PR[GP1:91,1] = PR[GP1:90,1] + -61.249;
   1:  PR[GP1:91,2] = PR[GP1:90,2] + 26.570;
   1:L PR[91] 10mm/sec CNT100;
   1:  PR[GP1:91,1] = PR[GP1:90,1] + -64.788;
   1:  PR[GP1:91,2] = PR[GP1:90,2] + 23.406;
   1:L PR[91] 10mm/sec CNT100;
   1:  PR[GP1:91,1] = PR[GP1:90,1] + -66.502;
   1:  PR[GP1:91,2] = PR[GP1:90,2] + 20.678;
   1:L PR[91] 10mm/sec CNT100;
   1:  PR[GP1:91,1] = PR[GP1:90,1] + -69.459;
   1:  PR[GP1:91,2] = PR[GP1:90,2] + 16.822;
   1:L PR[91] 10mm/sec CNT100;
   1:  PR[GP1:91,1] = PR[GP1:90,1] + -71.598;
   1:  PR[GP1:91,2] = PR[GP1:90,2] + 12.584;
   1:L PR[91] 10mm/sec CNT100;
   1:  PR[GP1:91,1] = PR[GP1:90,1] + -72.196;
   1:  PR[GP1:91,2] = PR[GP1:90,2] + 9.420;
   1:L PR[91] 10mm/sec CNT100;
   1:  PR[GP1:91,1] = PR[GP1:90,1] + -73.541;
   1:  PR[GP1:91,2] = PR[GP1:90,2] + 4.750;
   1:L PR[91] 10mm/sec CNT100;
   1:  PR[GP1:91,1] = PR[GP1:90,1] + -73.984;
   1:  PR[GP1:91,2] = PR[GP1:90,2] + 0.024;
   1:L PR[91] 10mm/sec CNT100;
   1:  PR[GP1:91,1] = PR[GP1:90,1] + -73.386;
   1:  PR[GP1:91,2] = PR[GP1:90,2] + -3.140;
   1:L PR[91] 10mm/sec CNT100;
   1:  PR[GP1:91,1] = PR[GP1:90,1] + -72.932;
   1:  PR[GP1:91,2] = PR[GP1:90,2] + -7.979;
   1:L PR[91] 10mm/sec CNT100;
   1:  PR[GP1:91,1] = PR[GP1:90,1] + -71.611;
   1:  PR[GP1:91,2] = PR[GP1:90,2] + -12.568;
   1:L PR[91] 10mm/sec CNT100;
   1:  PR[GP1:91,1] = PR[GP1:90,1] + -69.447;
   1:  PR[GP1:91,2] = PR[GP1:90,2] + -16.856;
   1:L PR[91] 10mm/sec CNT100;
   1:  PR[GP1:91,1] = PR[GP1:90,1] + -67.732;
   1:  PR[GP1:91,2] = PR[GP1:90,2] + -19.584;
   1:L PR[91] 10mm/sec CNT100;
   1:  PR[GP1:91,1] = PR[GP1:90,1] + -64.809;
   1:  PR[GP1:91,2] = PR[GP1:90,2] + -23.396;
   1:L PR[91] 10mm/sec CNT100;
   1:  PR[GP1:91,1] = PR[GP1:90,1] + -61.228;
   1:  PR[GP1:91,2] = PR[GP1:90,2] + -26.597;
   1:L PR[91] 10mm/sec CNT100;
   1:  PR[GP1:91,1] = PR[GP1:90,1] + -58.638;
   1:  PR[GP1:91,2] = PR[GP1:90,2] + -28.510;
   1:L PR[91] 10mm/sec CNT100;
   1:  PR[GP1:91,1] = PR[GP1:90,1] + -54.524;
   1:  PR[GP1:91,2] = PR[GP1:90,2] + -30.990;
   1:L PR[91] 10mm/sec CNT100;
   1:  PR[GP1:91,1] = PR[GP1:90,1] + -50.022;
   1:  PR[GP1:91,2] = PR[GP1:90,2] + -32.663;
   1:L PR[91] 10mm/sec CNT100;
   1:  PR[GP1:91,1] = PR[GP1:90,1] + -46.911;
   1:  PR[GP1:91,2] = PR[GP1:90,2] + -33.498;
   1:L PR[91] 10mm/sec CNT100;
   1:  PR[GP1:91,1] = PR[GP1:90,1] + -42.175;
   1:  PR[GP1:91,2] = PR[GP1:90,2] + -34.304;
   1:L PR[91] 10mm/sec CNT100;
   1:  PR[GP1:91,1] = PR[GP1:90,1] + -37.373;
   1:  PR[GP1:91,2] = PR[GP1:90,2] + -34.217;
   1:L PR[91] 10mm/sec CNT100;
   1:  PR[GP1:91,1] = PR[GP1:90,1] + -34.172;
   1:  PR[GP1:91,2] = PR[GP1:90,2] + -33.858;
   1:L PR[91] 10mm/sec CNT100;
   1:  PR[GP1:91,1] = PR[GP1:90,1] + -29.469;
   1:  PR[GP1:91,2] = PR[GP1:90,2] + -32.879;
   1:L PR[91] 10mm/sec CNT100;
   1:  PR[GP1:91,1] = PR[GP1:90,1] + -25.030;
   1:  PR[GP1:91,2] = PR[GP1:90,2] + -31.044;
   1:L PR[91] 10mm/sec CNT100;
   1:  PR[GP1:91,1] = PR[GP1:90,1] + -22.183;
   1:  PR[GP1:91,2] = PR[GP1:90,2] + -29.541;
   1:L PR[91] 10mm/sec CNT100;
   1:  PR[GP1:91,1] = PR[GP1:90,1] + -18.162;
   1:  PR[GP1:91,2] = PR[GP1:90,2] + -26.912;
   1:L PR[91] 10mm/sec CNT100;
   1:  PR[GP1:91,1] = PR[GP1:90,1] + -14.700;
   1:  PR[GP1:91,2] = PR[GP1:90,2] + -23.582;
   1:L PR[91] 10mm/sec CNT100;
   1:  PR[GP1:91,1] = PR[GP1:90,1] + -12.597;
   1:  PR[GP1:91,2] = PR[GP1:90,2] + -21.142;
   1:L PR[91] 10mm/sec CNT100;
   1:  PR[GP1:91,1] = PR[GP1:90,1] + -9.815;
   1:  PR[GP1:91,2] = PR[GP1:90,2] + -17.227;
   1:L PR[91] 10mm/sec CNT100;
   1:  PR[GP1:91,1] = PR[GP1:90,1] + -7.808;
   1:  PR[GP1:91,2] = PR[GP1:90,2] + -12.863;
   1:L PR[91] 10mm/sec CNT100;
   1:  PR[GP1:91,1] = PR[GP1:90,1] + -6.742;
   1:  PR[GP1:91,2] = PR[GP1:90,2] + -9.825;
   1:L PR[91] 10mm/sec CNT100;
   1:  PR[GP1:91,1] = PR[GP1:90,1] + -5.549;
   1:  PR[GP1:91,2] = PR[GP1:90,2] + -5.033;
   1:L PR[91] 10mm/sec CNT100;
   1:  PR[GP1:91,1] = PR[GP1:90,1] + -3.719;
   1:  PR[GP1:91,2] = PR[GP1:90,2] + -1.728;
   1:L PR[91] 10mm/sec CNT100;
   1:  PR[GP1:91,1] = PR[GP1:90,1] + -0.150;
   1:  PR[GP1:91,2] = PR[GP1:90,2] + -0.404;
   1:L PR[91] 10mm/sec CNT100;
   1:  PR[GP1:91,1] = PR[GP1:90,1] + 0.971;
   1:L PR[91] 10mm/sec CNT100;
   1:  PR[GP1:91,1] = PR[GP1:90,1] + 4.540;
   1:  PR[GP1:91,2] = PR[GP1:90,2] + -1.728;
   1:L PR[91] 10mm/sec CNT100;
   1:  PR[GP1:91,1] = PR[GP1:90,1] + 6.356;
   1:  PR[GP1:91,2] = PR[GP1:90,2] + -5.008;
   1:L PR[91] 10mm/sec CNT100;
   1:  PR[GP1:91,1] = PR[GP1:90,1] + 7.466;
   1:  PR[GP1:91,2] = PR[GP1:90,2] + -8.173;
   1:L PR[91] 10mm/sec CNT100;
   1:  PR[GP1:91,1] = PR[GP1:90,1] + 8.640;
   1:  PR[GP1:91,2] = PR[GP1:90,2] + -12.888;
   1:L PR[91] 10mm/sec CNT100;
   1:  PR[GP1:91,1] = PR[GP1:90,1] + 10.623;
   1:  PR[GP1:91,2] = PR[GP1:90,2] + -17.201;
   1:L PR[91] 10mm/sec CNT100;
   1:  PR[GP1:91,1] = PR[GP1:90,1] + 12.726;
   1:  PR[GP1:91,2] = PR[GP1:90,2] + -19.641;
   1:L PR[91] 10mm/sec CNT100;
   1:  PR[GP1:91,1] = PR[GP1:90,1] + 15.541;
   1:  PR[GP1:91,2] = PR[GP1:90,2] + -23.602;
   1:L PR[91] 10mm/sec CNT100;
   1:  PR[GP1:91,1] = PR[GP1:90,1] + 18.962;
   1:  PR[GP1:91,2] = PR[GP1:90,2] + -26.893;
   1:L PR[91] 10mm/sec CNT100;
   1:  PR[GP1:91,1] = PR[GP1:90,1] + 21.809;
   1:  PR[GP1:91,2] = PR[GP1:90,2] + -28.395;
   1:L PR[91] 10mm/sec CNT100;
   1:  PR[GP1:91,1] = PR[GP1:90,1] + 25.877;
   1:  PR[GP1:91,2] = PR[GP1:90,2] + -31.055;
   1:L PR[91] 10mm/sec CNT100;
   1:  PR[GP1:91,1] = PR[GP1:90,1] + 30.263;
   1:  PR[GP1:91,2] = PR[GP1:90,2] + -32.868;
   1:L PR[91] 10mm/sec CNT100;
   1:  PR[GP1:91,1] = PR[GP1:90,1] + 33.464;
   1:  PR[GP1:91,2] = PR[GP1:90,2] + -33.228;
   1:L PR[91] 10mm/sec CNT100;
   1:  PR[GP1:91,1] = PR[GP1:90,1] + 38.221;
   1:  PR[GP1:91,2] = PR[GP1:90,2] + -34.217;
   1:L PR[91] 10mm/sec CNT100;
   1:  PR[GP1:91,1] = PR[GP1:90,1] + 42.968;
   1:  PR[GP1:91,2] = PR[GP1:90,2] + -34.304;
   1:L PR[91] 10mm/sec CNT100;
   1:  PR[GP1:91,1] = PR[GP1:90,1] + 46.078;
   1:  PR[GP1:91,2] = PR[GP1:90,2] + -33.469;
   1:L PR[91] 10mm/sec CNT100;
   1:  PR[GP1:91,1] = PR[GP1:90,1] + 50.869;
   1:  PR[GP1:91,2] = PR[GP1:90,2] + -32.653;
   1:L PR[91] 10mm/sec CNT100;
   1:  PR[GP1:91,1] = PR[GP1:90,1] + 55.319;
   1:  PR[GP1:91,2] = PR[GP1:90,2] + -31.000;
   1:L PR[91] 10mm/sec CNT100;
   1:  PR[GP1:91,1] = PR[GP1:90,1] + 57.909;
   1:  PR[GP1:91,2] = PR[GP1:90,2] + -29.088;
   1:L PR[91] 10mm/sec CNT100;
   1:  PR[GP1:91,1] = PR[GP1:90,1] + 62.070;
   1:  PR[GP1:91,2] = PR[GP1:90,2] + -26.579;
   1:L PR[91] 10mm/sec CNT100;
   1:  PR[GP1:91,1] = PR[GP1:90,1] + 65.609;
   1:  PR[GP1:91,2] = PR[GP1:90,2] + -23.415;
   1:L PR[91] 10mm/sec CNT100;
   1:  PR[GP1:91,1] = PR[GP1:90,1] + 67.322;
   1:  PR[GP1:91,2] = PR[GP1:90,2] + -20.687;
   1:L PR[91] 10mm/sec CNT100;
   1:  PR[GP1:91,1] = PR[GP1:90,1] + 70.280;
   1:  PR[GP1:91,2] = PR[GP1:90,2] + -16.831;
   1:L PR[91] 10mm/sec CNT100;
   1:  PR[GP1:91,1] = PR[GP1:90,1] + 72.418;
   1:  PR[GP1:91,2] = PR[GP1:90,2] + -12.593;
   1:L PR[91] 10mm/sec CNT100;
   1:  PR[GP1:91,1] = PR[GP1:90,1] + 73.017;
   1:  PR[GP1:91,2] = PR[GP1:90,2] + -9.429;
   1:L PR[91] 10mm/sec CNT100;
   1:  PR[GP1:91,1] = PR[GP1:90,1] + 74.362;
   1:  PR[GP1:91,2] = PR[GP1:90,2] + -4.759;
   1:L PR[91] 10mm/sec CNT100;
   1:  PR[GP1:91,1] = PR[GP1:90,1] + 74.805;
   1:  PR[GP1:91,2] = PR[GP1:90,2] + -0.033;
   1:L PR[91] 10mm/sec CNT100;
   1:  PR[GP1:91,1] = PR[GP1:90,1] + 74.206;
   1:  PR[GP1:91,2] = PR[GP1:90,2] + 3.132;
   1:L PR[91] 10mm/sec CNT100;
   1:  PR[GP1:91,1] = PR[GP1:90,1] + 73.753;
   1:  PR[GP1:91,2] = PR[GP1:90,2] + 7.970;
   1:L PR[91] 10mm/sec CNT100;
   1:  PR[GP1:91,1] = PR[GP1:90,1] + 72.431;
   1:  PR[GP1:91,2] = PR[GP1:90,2] + 12.559;
   1:L PR[91] 10mm/sec CNT100;
   1:  PR[GP1:91,1] = PR[GP1:90,1] + 70.267;
   1:  PR[GP1:91,2] = PR[GP1:90,2] + 16.847;
   1:L PR[91] 10mm/sec CNT100;
   1:  PR[GP1:91,1] = PR[GP1:90,1] + 68.553;
   1:  PR[GP1:91,2] = PR[GP1:90,2] + 19.575;
   1:L PR[91] 10mm/sec CNT100;
   1:  PR[GP1:91,1] = PR[GP1:90,1] + 65.630;
   1:  PR[GP1:91,2] = PR[GP1:90,2] + 23.387;
   1:L PR[91] 10mm/sec CNT100;
   1:  PR[GP1:91,1] = PR[GP1:90,1] + 62.049;
   1:  PR[GP1:91,2] = PR[GP1:90,2] + 26.589;
   1:L PR[91] 10mm/sec CNT100;
   1:  PR[GP1:91,1] = PR[GP1:90,1] + 59.459;
   1:  PR[GP1:91,2] = PR[GP1:90,2] + 28.501;
   1:L PR[91] 10mm/sec CNT100;
   1:  PR[GP1:91,1] = PR[GP1:90,1] + 55.345;
   1:  PR[GP1:91,2] = PR[GP1:90,2] + 30.981;
   1:L PR[91] 10mm/sec CNT100;
   1:  PR[GP1:91,1] = PR[GP1:90,1] + 50.842;
   1:  PR[GP1:91,2] = PR[GP1:90,2] + 32.654;
   1:L PR[91] 10mm/sec CNT100;
   1:  PR[GP1:91,1] = PR[GP1:90,1] + 47.731;
   1:  PR[GP1:91,2] = PR[GP1:90,2] + 33.489;
   1:L PR[91] 10mm/sec CNT100;
   1:  PR[GP1:91,1] = PR[GP1:90,1] + 42.996;
   1:  PR[GP1:91,2] = PR[GP1:90,2] + 34.295;
   1:L PR[91] 10mm/sec CNT100;
   1:  PR[GP1:91,1] = PR[GP1:90,1] + 38.193;
   1:  PR[GP1:91,2] = PR[GP1:90,2] + 34.208;
   1:L PR[91] 10mm/sec CNT100;
   1:  PR[GP1:91,1] = PR[GP1:90,1] + 34.992;
   1:  PR[GP1:91,2] = PR[GP1:90,2] + 33.849;
   1:L PR[91] 10mm/sec CNT100;
   1:  PR[GP1:91,1] = PR[GP1:90,1] + 30.290;
   1:  PR[GP1:91,2] = PR[GP1:90,2] + 32.870;
   1:L PR[91] 10mm/sec CNT100;
   1:  PR[GP1:91,1] = PR[GP1:90,1] + 25.851;
   1:  PR[GP1:91,2] = PR[GP1:90,2] + 31.035;
   1:L PR[91] 10mm/sec CNT100;
   1:  PR[GP1:91,1] = PR[GP1:90,1] + 23.003;
   1:  PR[GP1:91,2] = PR[GP1:90,2] + 29.532;
   1:L PR[91] 10mm/sec CNT100;
   1:  PR[GP1:91,1] = PR[GP1:90,1] + 18.983;
   1:  PR[GP1:91,2] = PR[GP1:90,2] + 26.904;
   1:L PR[91] 10mm/sec CNT100;
   1:  PR[GP1:91,1] = PR[GP1:90,1] + 15.521;
   1:  PR[GP1:91,2] = PR[GP1:90,2] + 23.574;
   1:L PR[91] 10mm/sec CNT100;
   1:  PR[GP1:91,1] = PR[GP1:90,1] + 13.418;
   1:  PR[GP1:91,2] = PR[GP1:90,2] + 21.133;
   1:L PR[91] 10mm/sec CNT100;
   1:  PR[GP1:91,1] = PR[GP1:90,1] + 10.635;
   1:  PR[GP1:91,2] = PR[GP1:90,2] + 17.218;
   1:L PR[91] 10mm/sec CNT100;
   1:  PR[GP1:91,1] = PR[GP1:90,1] + 8.629;
   1:  PR[GP1:91,2] = PR[GP1:90,2] + 12.854;
   1:L PR[91] 10mm/sec CNT100;
   1:  PR[GP1:91,1] = PR[GP1:90,1] + 7.563;
   1:  PR[GP1:91,2] = PR[GP1:90,2] + 9.816;
   1:L PR[91] 10mm/sec CNT100;
   1:  PR[GP1:91,1] = PR[GP1:90,1] + 6.369;
   1:  PR[GP1:91,2] = PR[GP1:90,2] + 5.024;
   1:L PR[91] 10mm/sec CNT100;
   1:  PR[GP1:91,1] = PR[GP1:90,1] + 4.540;
   1:  PR[GP1:91,2] = PR[GP1:90,2] + 1.719;
   1:L PR[91] 10mm/sec CNT100;
   1:  PR[GP1:91,1] = PR[GP1:90,1] + 0.971;
   1:  PR[GP1:91,2] = PR[GP1:90,2] + 0.396;
   1:L PR[91] 10mm/sec CNT100;
   1:  PR[GP1:91,1] = PR[GP1:90,1] + -0.150;
   1:L PR[91] 10mm/sec CNT100;
   1:  PR[GP1:91,1] = PR[GP1:90,1] + -3.719;
   1:  PR[GP1:91,2] = PR[GP1:90,2] + 1.719;
   1:  PR[GP1:91,3] = PR[GP1:90,3] + 7.980;
   1:L PR[91] 10mm/sec CNT100;
   1:  PR[GP1:91,1] = PR[GP1:90,1] + -5.535;
   1:  PR[GP1:91,2] = PR[GP1:90,2] + 4.999;
   1:L PR[91] 10mm/sec CNT100;
   1:  PR[GP1:91,1] = PR[GP1:90,1] + -5.930;
   1:  PR[GP1:91,2] = PR[GP1:90,2] + 6.124;
   1:L PR[91] 10mm/sec CNT100;
   1:  PR[GP1:91,1] = PR[GP1:90,1] + -7.366;
   1:  PR[GP1:91,2] = PR[GP1:90,2] + 11.893;
   1:L PR[91] 10mm/sec CNT100;
   1:  PR[GP1:91,1] = PR[GP1:90,1] + -9.803;
   1:  PR[GP1:91,2] = PR[GP1:90,2] + 17.193;
   1:L PR[91] 10mm/sec CNT100;
   1:  PR[GP1:91,1] = PR[GP1:90,1] + -10.494;
   1:  PR[GP1:91,2] = PR[GP1:90,2] + 17.994;
   1:L PR[91] 10mm/sec CNT100;
   1:  PR[GP1:91,1] = PR[GP1:90,1] + -13.938;
   1:  PR[GP1:91,2] = PR[GP1:90,2] + 22.841;
   1:L PR[91] 10mm/sec CNT100;
   1:  PR[GP1:91,1] = PR[GP1:90,1] + -18.142;
   1:  PR[GP1:91,2] = PR[GP1:90,2] + 26.884;
   1:L PR[91] 10mm/sec CNT100;
   1:  PR[GP1:91,1] = PR[GP1:90,1] + -19.077;
   1:  PR[GP1:91,2] = PR[GP1:90,2] + 27.378;
   1:L PR[91] 10mm/sec CNT100;
   1:  PR[GP1:91,1] = PR[GP1:90,1] + -24.053;
   1:  PR[GP1:91,2] = PR[GP1:90,2] + 30.631;
   1:L PR[91] 10mm/sec CNT100;
   1:  PR[GP1:91,1] = PR[GP1:90,1] + -29.444;
   1:  PR[GP1:91,2] = PR[GP1:90,2] + 32.860;
   1:L PR[91] 10mm/sec CNT100;
   1:  PR[GP1:91,1] = PR[GP1:90,1] + -30.495;
   1:  PR[GP1:91,2] = PR[GP1:90,2] + 32.978;
   1:L PR[91] 10mm/sec CNT100;
   1:  PR[GP1:91,1] = PR[GP1:90,1] + -36.316;
   1:  PR[GP1:91,2] = PR[GP1:90,2] + 34.189;
   1:L PR[91] 10mm/sec CNT100;
   1:  PR[GP1:91,1] = PR[GP1:90,1] + -42.148;
   1:  PR[GP1:91,2] = PR[GP1:90,2] + 34.295;
   1:L PR[91] 10mm/sec CNT100;
   1:  PR[GP1:91,1] = PR[GP1:90,1] + -43.169;
   1:  PR[GP1:91,2] = PR[GP1:90,2] + 34.021;
   1:L PR[91] 10mm/sec CNT100;
   1:  PR[GP1:91,1] = PR[GP1:90,1] + -49.031;
   1:  PR[GP1:91,2] = PR[GP1:90,2] + 33.022;
   1:L PR[91] 10mm/sec CNT100;
   1:  PR[GP1:91,1] = PR[GP1:90,1] + -54.498;
   1:  PR[GP1:91,2] = PR[GP1:90,2] + 30.991;
   1:L PR[91] 10mm/sec CNT100;
   1:  PR[GP1:91,1] = PR[GP1:90,1] + -55.349;
   1:  PR[GP1:91,2] = PR[GP1:90,2] + 30.363;
   1:L PR[91] 10mm/sec CNT100;
   1:  PR[GP1:91,1] = PR[GP1:90,1] + -60.440;
   1:  PR[GP1:91,2] = PR[GP1:90,2] + 27.293;
   1:L PR[91] 10mm/sec CNT100;
   1:  PR[GP1:91,1] = PR[GP1:90,1] + -64.789;
   1:  PR[GP1:91,2] = PR[GP1:90,2] + 23.405;
   1:L PR[91] 10mm/sec CNT100;
   1:  PR[GP1:91,1] = PR[GP1:90,1] + -65.352;
   1:  PR[GP1:91,2] = PR[GP1:90,2] + 22.509;
   1:L PR[91] 10mm/sec CNT100;
   1:  PR[GP1:91,1] = PR[GP1:90,1] + -68.970;
   1:  PR[GP1:91,2] = PR[GP1:90,2] + 17.791;
   1:L PR[91] 10mm/sec CNT100;
   1:  PR[GP1:91,1] = PR[GP1:90,1] + -71.598;
   1:  PR[GP1:91,2] = PR[GP1:90,2] + 12.584;
   1:L PR[91] 10mm/sec CNT100;
   1:  PR[GP1:91,1] = PR[GP1:90,1] + -71.794;
   1:  PR[GP1:91,2] = PR[GP1:90,2] + 11.545;
   1:L PR[91] 10mm/sec CNT100;
   1:  PR[GP1:91,1] = PR[GP1:90,1] + -73.440;
   1:  PR[GP1:91,2] = PR[GP1:90,2] + 5.831;
   1:L PR[91] 10mm/sec CNT100;
   1:  PR[GP1:91,1] = PR[GP1:90,1] + -73.984;
   1:  PR[GP1:91,2] = PR[GP1:90,2] + 0.024;
   1:L PR[91] 10mm/sec CNT100;
   1:  PR[GP1:91,1] = PR[GP1:90,1] + -73.788;
   1:  PR[GP1:91,2] = PR[GP1:90,2] + -1.015;
   1:L PR[91] 10mm/sec CNT100;
   1:  PR[GP1:91,1] = PR[GP1:90,1] + -73.233;
   1:  PR[GP1:91,2] = PR[GP1:90,2] + -6.935;
   1:L PR[91] 10mm/sec CNT100;
   1:  PR[GP1:91,1] = PR[GP1:90,1] + -71.611;
   1:  PR[GP1:91,2] = PR[GP1:90,2] + -12.567;
   1:L PR[91] 10mm/sec CNT100;
   1:  PR[GP1:91,1] = PR[GP1:90,1] + -68.957;
   1:  PR[GP1:91,2] = PR[GP1:90,2] + -17.825;
   1:L PR[91] 10mm/sec CNT100;
   1:  PR[GP1:91,1] = PR[GP1:90,1] + -68.394;
   1:  PR[GP1:91,2] = PR[GP1:90,2] + -18.722;
   1:L PR[91] 10mm/sec CNT100;
   1:  PR[GP1:91,1] = PR[GP1:90,1] + -64.810;
   1:  PR[GP1:91,2] = PR[GP1:90,2] + -23.395;
   1:L PR[91] 10mm/sec CNT100;
   1:  PR[GP1:91,1] = PR[GP1:90,1] + -60.420;
   1:  PR[GP1:91,2] = PR[GP1:90,2] + -27.321;
   1:L PR[91] 10mm/sec CNT100;
   1:  PR[GP1:91,1] = PR[GP1:90,1] + -59.569;
   1:  PR[GP1:91,2] = PR[GP1:90,2] + -27.949;
   1:L PR[91] 10mm/sec CNT100;
   1:  PR[GP1:91,1] = PR[GP1:90,1] + -54.525;
   1:  PR[GP1:91,2] = PR[GP1:90,2] + -30.990;
   1:L PR[91] 10mm/sec CNT100;
   1:  PR[GP1:91,1] = PR[GP1:90,1] + -49.004;
   1:  PR[GP1:91,2] = PR[GP1:90,2] + -33.041;
   1:L PR[91] 10mm/sec CNT100;
   1:  PR[GP1:91,1] = PR[GP1:90,1] + -47.982;
   1:  PR[GP1:91,2] = PR[GP1:90,2] + -33.315;
   1:L PR[91] 10mm/sec CNT100;
   1:  PR[GP1:91,1] = PR[GP1:90,1] + -42.176;
   1:  PR[GP1:91,2] = PR[GP1:90,2] + -34.304;
   1:L PR[91] 10mm/sec CNT100;
   1:  PR[GP1:91,1] = PR[GP1:90,1] + -36.288;
   1:  PR[GP1:91,2] = PR[GP1:90,2] + -34.197;
   1:L PR[91] 10mm/sec CNT100;
   1:  PR[GP1:91,1] = PR[GP1:90,1] + -35.236;
   1:  PR[GP1:91,2] = PR[GP1:90,2] + -34.079;
   1:L PR[91] 10mm/sec CNT100;
   1:  PR[GP1:91,1] = PR[GP1:90,1] + -29.470;
   1:  PR[GP1:91,2] = PR[GP1:90,2] + -32.880;
   1:L PR[91] 10mm/sec CNT100;
   1:  PR[GP1:91,1] = PR[GP1:90,1] + -24.027;
   1:  PR[GP1:91,2] = PR[GP1:90,2] + -30.629;
   1:L PR[91] 10mm/sec CNT100;
   1:  PR[GP1:91,1] = PR[GP1:90,1] + -23.092;
   1:  PR[GP1:91,2] = PR[GP1:90,2] + -30.135;
   1:L PR[91] 10mm/sec CNT100;
   1:  PR[GP1:91,1] = PR[GP1:90,1] + -18.163;
   1:  PR[GP1:91,2] = PR[GP1:90,2] + -26.913;
   1:L PR[91] 10mm/sec CNT100;
   1:  PR[GP1:91,1] = PR[GP1:90,1] + -13.918;
   1:  PR[GP1:91,2] = PR[GP1:90,2] + -22.830;
   1:L PR[91] 10mm/sec CNT100;
   1:  PR[GP1:91,1] = PR[GP1:90,1] + -13.227;
   1:  PR[GP1:91,2] = PR[GP1:90,2] + -22.028;
   1:L PR[91] 10mm/sec CNT100;
   1:  PR[GP1:91,1] = PR[GP1:90,1] + -9.815;
   1:  PR[GP1:91,2] = PR[GP1:90,2] + -17.228;
   1:L PR[91] 10mm/sec CNT100;
   1:  PR[GP1:91,1] = PR[GP1:90,1] + -7.355;
   1:  PR[GP1:91,2] = PR[GP1:90,2] + -11.877;
   1:L PR[91] 10mm/sec CNT100;
   1:  PR[GP1:91,1] = PR[GP1:90,1] + -7.005;
   1:  PR[GP1:91,2] = PR[GP1:90,2] + -10.879;
   1:L PR[91] 10mm/sec CNT100;
   1:  PR[GP1:91,1] = PR[GP1:90,1] + -5.549;
   1:  PR[GP1:91,2] = PR[GP1:90,2] + -5.033;
   1:L PR[91] 10mm/sec CNT100;
   1:  PR[GP1:91,1] = PR[GP1:90,1] + -3.719;
   1:  PR[GP1:91,2] = PR[GP1:90,2] + -1.728;
   1:L PR[91] 10mm/sec CNT100;
   1:  PR[GP1:91,1] = PR[GP1:90,1] + -0.150;
   1:  PR[GP1:91,2] = PR[GP1:90,2] + -0.404;
   1:L PR[91] 10mm/sec CNT100;
   1:  PR[GP1:91,1] = PR[GP1:90,1] + 0.971;
   1:L PR[91] 10mm/sec CNT100;
   1:  PR[GP1:91,1] = PR[GP1:90,1] + 4.540;
   1:  PR[GP1:91,2] = PR[GP1:90,2] + -1.728;
   1:L PR[91] 10mm/sec CNT100;
   1:  PR[GP1:91,1] = PR[GP1:90,1] + 6.356;
   1:  PR[GP1:91,2] = PR[GP1:90,2] + -5.008;
   1:L PR[91] 10mm/sec CNT100;
   1:  PR[GP1:91,1] = PR[GP1:90,1] + 6.750;
   1:  PR[GP1:91,2] = PR[GP1:90,2] + -6.133;
   1:L PR[91] 10mm/sec CNT100;
   1:  PR[GP1:91,1] = PR[GP1:90,1] + 8.187;
   1:  PR[GP1:91,2] = PR[GP1:90,2] + -11.902;
   1:L PR[91] 10mm/sec CNT100;
   1:  PR[GP1:91,1] = PR[GP1:90,1] + 10.624;
   1:  PR[GP1:91,2] = PR[GP1:90,2] + -17.202;
   1:L PR[91] 10mm/sec CNT100;
   1:  PR[GP1:91,1] = PR[GP1:90,1] + 11.314;
   1:  PR[GP1:91,2] = PR[GP1:90,2] + -18.003;
   1:L PR[91] 10mm/sec CNT100;
   1:  PR[GP1:91,1] = PR[GP1:90,1] + 14.759;
   1:  PR[GP1:91,2] = PR[GP1:90,2] + -22.849;
   1:L PR[91] 10mm/sec CNT100;
   1:  PR[GP1:91,1] = PR[GP1:90,1] + 18.963;
   1:  PR[GP1:91,2] = PR[GP1:90,2] + -26.893;
   1:L PR[91] 10mm/sec CNT100;
   1:  PR[GP1:91,1] = PR[GP1:90,1] + 19.897;
   1:  PR[GP1:91,2] = PR[GP1:90,2] + -27.386;
   1:L PR[91] 10mm/sec CNT100;
   1:  PR[GP1:91,1] = PR[GP1:90,1] + 24.874;
   1:  PR[GP1:91,2] = PR[GP1:90,2] + -30.640;
   1:L PR[91] 10mm/sec CNT100;
   1:  PR[GP1:91,1] = PR[GP1:90,1] + 30.265;
   1:  PR[GP1:91,2] = PR[GP1:90,2] + -32.869;
   1:L PR[91] 10mm/sec CNT100;
   1:  PR[GP1:91,1] = PR[GP1:90,1] + 31.315;
   1:  PR[GP1:91,2] = PR[GP1:90,2] + -32.987;
   1:L PR[91] 10mm/sec CNT100;
   1:  PR[GP1:91,1] = PR[GP1:90,1] + 37.136;
   1:  PR[GP1:91,2] = PR[GP1:90,2] + -34.198;
   1:L PR[91] 10mm/sec CNT100;
   1:  PR[GP1:91,1] = PR[GP1:90,1] + 42.969;
   1:  PR[GP1:91,2] = PR[GP1:90,2] + -34.304;
   1:L PR[91] 10mm/sec CNT100;
   1:  PR[GP1:91,1] = PR[GP1:90,1] + 43.990;
   1:  PR[GP1:91,2] = PR[GP1:90,2] + -34.030;
   1:L PR[91] 10mm/sec CNT100;
   1:  PR[GP1:91,1] = PR[GP1:90,1] + 49.851;
   1:  PR[GP1:91,2] = PR[GP1:90,2] + -33.031;
   1:L PR[91] 10mm/sec CNT100;
   1:  PR[GP1:91,1] = PR[GP1:90,1] + 55.319;
   1:  PR[GP1:91,2] = PR[GP1:90,2] + -31.000;
   1:L PR[91] 10mm/sec CNT100;
   1:  PR[GP1:91,1] = PR[GP1:90,1] + 56.170;
   1:  PR[GP1:91,2] = PR[GP1:90,2] + -30.372;
   1:L PR[91] 10mm/sec CNT100;
   1:  PR[GP1:91,1] = PR[GP1:90,1] + 61.261;
   1:  PR[GP1:91,2] = PR[GP1:90,2] + -27.302;
   1:L PR[91] 10mm/sec CNT100;
   1:  PR[GP1:91,1] = PR[GP1:90,1] + 65.609;
   1:  PR[GP1:91,2] = PR[GP1:90,2] + -23.414;
   1:L PR[91] 10mm/sec CNT100;
   1:  PR[GP1:91,1] = PR[GP1:90,1] + 66.172;
   1:  PR[GP1:91,2] = PR[GP1:90,2] + -22.518;
   1:L PR[91] 10mm/sec CNT100;
   1:  PR[GP1:91,1] = PR[GP1:90,1] + 69.791;
   1:  PR[GP1:91,2] = PR[GP1:90,2] + -17.800;
   1:L PR[91] 10mm/sec CNT100;
   1:  PR[GP1:91,1] = PR[GP1:90,1] + 72.419;
   1:  PR[GP1:91,2] = PR[GP1:90,2] + -12.593;
   1:L PR[91] 10mm/sec CNT100;
   1:  PR[GP1:91,1] = PR[GP1:90,1] + 72.615;
   1:  PR[GP1:91,2] = PR[GP1:90,2] + -11.554;
   1:L PR[91] 10mm/sec CNT100;
   1:  PR[GP1:91,1] = PR[GP1:90,1] + 74.261;
   1:  PR[GP1:91,2] = PR[GP1:90,2] + -5.840;
   1:L PR[91] 10mm/sec CNT100;
   1:  PR[GP1:91,1] = PR[GP1:90,1] + 74.805;
   1:  PR[GP1:91,2] = PR[GP1:90,2] + -0.033;
   1:L PR[91] 10mm/sec CNT100;
   1:  PR[GP1:91,1] = PR[GP1:90,1] + 74.608;
   1:  PR[GP1:91,2] = PR[GP1:90,2] + 1.006;
   1:L PR[91] 10mm/sec CNT100;
   1:  PR[GP1:91,1] = PR[GP1:90,1] + 74.053;
   1:  PR[GP1:91,2] = PR[GP1:90,2] + 6.926;
   1:L PR[91] 10mm/sec CNT100;
   1:  PR[GP1:91,1] = PR[GP1:90,1] + 72.431;
   1:  PR[GP1:91,2] = PR[GP1:90,2] + 12.559;
   1:L PR[91] 10mm/sec CNT100;
   1:  PR[GP1:91,1] = PR[GP1:90,1] + 69.778;
   1:  PR[GP1:91,2] = PR[GP1:90,2] + 17.817;
   1:L PR[91] 10mm/sec CNT100;
   1:  PR[GP1:91,1] = PR[GP1:90,1] + 69.215;
   1:  PR[GP1:91,2] = PR[GP1:90,2] + 18.713;
   1:L PR[91] 10mm/sec CNT100;
   1:  PR[GP1:91,1] = PR[GP1:90,1] + 65.631;
   1:  PR[GP1:91,2] = PR[GP1:90,2] + 23.386;
   1:L PR[91] 10mm/sec CNT100;
   1:  PR[GP1:91,1] = PR[GP1:90,1] + 61.240;
   1:  PR[GP1:91,2] = PR[GP1:90,2] + 27.312;
   1:L PR[91] 10mm/sec CNT100;
   1:  PR[GP1:91,1] = PR[GP1:90,1] + 60.389;
   1:  PR[GP1:91,2] = PR[GP1:90,2] + 27.940;
   1:L PR[91] 10mm/sec CNT100;
   1:  PR[GP1:91,1] = PR[GP1:90,1] + 55.346;
   1:  PR[GP1:91,2] = PR[GP1:90,2] + 30.981;
   1:L PR[91] 10mm/sec CNT100;
   1:  PR[GP1:91,1] = PR[GP1:90,1] + 49.825;
   1:  PR[GP1:91,2] = PR[GP1:90,2] + 33.032;
   1:L PR[91] 10mm/sec CNT100;
   1:  PR[GP1:91,1] = PR[GP1:90,1] + 48.803;
   1:  PR[GP1:91,2] = PR[GP1:90,2] + 33.306;
   1:L PR[91] 10mm/sec CNT100;
   1:  PR[GP1:91,1] = PR[GP1:90,1] + 42.997;
   1:  PR[GP1:91,2] = PR[GP1:90,2] + 34.295;
   1:L PR[91] 10mm/sec CNT100;
   1:  PR[GP1:91,1] = PR[GP1:90,1] + 37.108;
   1:  PR[GP1:91,2] = PR[GP1:90,2] + 34.188;
   1:L PR[91] 10mm/sec CNT100;
   1:  PR[GP1:91,1] = PR[GP1:90,1] + 36.057;
   1:  PR[GP1:91,2] = PR[GP1:90,2] + 34.070;
   1:L PR[91] 10mm/sec CNT100;
   1:  PR[GP1:91,1] = PR[GP1:90,1] + 30.291;
   1:  PR[GP1:91,2] = PR[GP1:90,2] + 32.871;
   1:L PR[91] 10mm/sec CNT100;
   1:  PR[GP1:91,1] = PR[GP1:90,1] + 24.848;
   1:  PR[GP1:91,2] = PR[GP1:90,2] + 30.620;
   1:L PR[91] 10mm/sec CNT100;
   1:  PR[GP1:91,1] = PR[GP1:90,1] + 23.913;
   1:  PR[GP1:91,2] = PR[GP1:90,2] + 30.127;
   1:L PR[91] 10mm/sec CNT100;
   1:  PR[GP1:91,1] = PR[GP1:90,1] + 18.983;
   1:  PR[GP1:91,2] = PR[GP1:90,2] + 26.904;
   1:L PR[91] 10mm/sec CNT100;
   1:  PR[GP1:91,1] = PR[GP1:90,1] + 14.738;
   1:  PR[GP1:91,2] = PR[GP1:90,2] + 22.821;
   1:L PR[91] 10mm/sec CNT100;
   1:  PR[GP1:91,1] = PR[GP1:90,1] + 14.048;
   1:  PR[GP1:91,2] = PR[GP1:90,2] + 22.020;
   1:L PR[91] 10mm/sec CNT100;
   1:  PR[GP1:91,1] = PR[GP1:90,1] + 10.636;
   1:  PR[GP1:91,2] = PR[GP1:90,2] + 17.219;
   1:L PR[91] 10mm/sec CNT100;
   1:  PR[GP1:91,1] = PR[GP1:90,1] + 8.175;
   1:  PR[GP1:91,2] = PR[GP1:90,2] + 11.868;
   1:L PR[91] 10mm/sec CNT100;
   1:  PR[GP1:91,1] = PR[GP1:90,1] + 7.825;
   1:  PR[GP1:91,2] = PR[GP1:90,2] + 10.870;
   1:L PR[91] 10mm/sec CNT100;
   1:  PR[GP1:91,1] = PR[GP1:90,1] + 6.369;
   1:  PR[GP1:91,2] = PR[GP1:90,2] + 5.024;
   1:L PR[91] 10mm/sec CNT100;
   1:  PR[GP1:91,1] = PR[GP1:90,1] + 4.540;
   1:  PR[GP1:91,2] = PR[GP1:90,2] + 1.719;
   1:L PR[91] 10mm/sec CNT100;
   1:  PR[GP1:91,1] = PR[GP1:90,1] + 0.971;
   1:  PR[GP1:91,2] = PR[GP1:90,2] + 0.396;
   1:L PR[91] 10mm/sec CNT100;
   1:  PR[GP1:91,1] = PR[GP1:90,1] + -0.150;
   1:L PR[91] 10mm/sec CNT100;
   1:  PR[GP1:91,1] = PR[GP1:90,1] + -3.672;
   1:  PR[GP1:91,2] = PR[GP1:90,2] + 1.720;
   1:  PR[GP1:91,3] = PR[GP1:90,3] + 9.310;
   1:L PR[91] 10mm/sec CNT100;
   1:  PR[GP1:91,1] = PR[GP1:90,1] + -5.290;
   1:  PR[GP1:91,2] = PR[GP1:90,2] + 4.642;
   1:L PR[91] 10mm/sec CNT100;
   1:  PR[GP1:91,1] = PR[GP1:90,1] + -5.803;
   1:  PR[GP1:91,2] = PR[GP1:90,2] + 5.459;
   1:L PR[91] 10mm/sec CNT100;
   1:  PR[GP1:91,1] = PR[GP1:90,1] + -5.631;
   1:  PR[GP1:91,2] = PR[GP1:90,2] + 5.556;
   1:L PR[91] 10mm/sec CNT100;
   1:  PR[GP1:91,1] = PR[GP1:90,1] + -6.949;
   1:  PR[GP1:91,2] = PR[GP1:90,2] + 10.845;
   1:L PR[91] 10mm/sec CNT100;
   1:  PR[GP1:91,1] = PR[GP1:90,1] + -7.262;
   1:  PR[GP1:91,2] = PR[GP1:90,2] + 11.790;
   1:L PR[91] 10mm/sec CNT100;
   1:  PR[GP1:91,1] = PR[GP1:90,1] + -9.713;
   1:  PR[GP1:91,2] = PR[GP1:90,2] + 17.121;
   1:L PR[91] 10mm/sec CNT100;
   1:  PR[GP1:91,1] = PR[GP1:90,1] + -13.125;
   1:  PR[GP1:91,2] = PR[GP1:90,2] + 21.922;
   1:L PR[91] 10mm/sec CNT100;
   1:  PR[GP1:91,1] = PR[GP1:90,1] + -13.701;
   1:  PR[GP1:91,2] = PR[GP1:90,2] + 22.676;
   1:L PR[91] 10mm/sec CNT100;
   1:  PR[GP1:91,1] = PR[GP1:90,1] + -17.946;
   1:  PR[GP1:91,2] = PR[GP1:90,2] + 26.759;
   1:L PR[91] 10mm/sec CNT100;
   1:  PR[GP1:91,1] = PR[GP1:90,1] + -23.657;
   1:  PR[GP1:91,2] = PR[GP1:90,2] + 30.500;
   1:L PR[91] 10mm/sec CNT100;
   1:  PR[GP1:91,1] = PR[GP1:90,1] + -29.129;
   1:  PR[GP1:91,2] = PR[GP1:90,2] + 32.763;
   1:L PR[91] 10mm/sec CNT100;
   1:  PR[GP1:91,1] = PR[GP1:90,1] + -34.996;
   1:  PR[GP1:91,2] = PR[GP1:90,2] + 33.983;
   1:L PR[91] 10mm/sec CNT100;
   1:  PR[GP1:91,1] = PR[GP1:90,1] + -35.796;
   1:  PR[GP1:91,2] = PR[GP1:90,2] + 34.191;
   1:L PR[91] 10mm/sec CNT100;
   1:  PR[GP1:91,1] = PR[GP1:90,1] + -41.772;
   1:  PR[GP1:91,2] = PR[GP1:90,2] + 34.299;
   1:L PR[91] 10mm/sec CNT100;
   1:  PR[GP1:91,1] = PR[GP1:90,1] + -42.496;
   1:  PR[GP1:91,2] = PR[GP1:90,2] + 34.245;
   1:L PR[91] 10mm/sec CNT100;
   1:  PR[GP1:91,1] = PR[GP1:90,1] + -48.437;
   1:  PR[GP1:91,2] = PR[GP1:90,2] + 33.232;
   1:L PR[91] 10mm/sec CNT100;
   1:  PR[GP1:91,1] = PR[GP1:90,1] + -54.099;
   1:  PR[GP1:91,2] = PR[GP1:90,2] + 31.129;
   1:L PR[91] 10mm/sec CNT100;
   1:  PR[GP1:91,1] = PR[GP1:90,1] + -54.718;
   1:  PR[GP1:91,2] = PR[GP1:90,2] + 30.862;
   1:L PR[91] 10mm/sec CNT100;
   1:  PR[GP1:91,1] = PR[GP1:90,1] + -59.893;
   1:  PR[GP1:91,2] = PR[GP1:90,2] + 27.742;
   1:L PR[91] 10mm/sec CNT100;
   1:  PR[GP1:91,1] = PR[GP1:90,1] + -64.896;
   1:  PR[GP1:91,2] = PR[GP1:90,2] + 23.260;
   1:L PR[91] 10mm/sec CNT100;
   1:  PR[GP1:91,1] = PR[GP1:90,1] + -68.576;
   1:  PR[GP1:91,2] = PR[GP1:90,2] + 18.461;
   1:L PR[91] 10mm/sec CNT100;
   1:  PR[GP1:91,1] = PR[GP1:90,1] + -71.331;
   1:  PR[GP1:91,2] = PR[GP1:90,2] + 13.004;
   1:L PR[91] 10mm/sec CNT100;
   1:  PR[GP1:91,1] = PR[GP1:90,1] + -71.619;
   1:  PR[GP1:91,2] = PR[GP1:90,2] + 12.474;
   1:L PR[91] 10mm/sec CNT100;
   1:  PR[GP1:91,1] = PR[GP1:90,1] + -73.293;
   1:  PR[GP1:91,2] = PR[GP1:90,2] + 6.660;
   1:L PR[91] 10mm/sec CNT100;
   1:  PR[GP1:91,1] = PR[GP1:90,1] + -73.866;
   1:  PR[GP1:91,2] = PR[GP1:90,2] + 0.550;
   1:L PR[91] 10mm/sec CNT100;
   1:  PR[GP1:91,1] = PR[GP1:90,1] + -73.962;
   1:  PR[GP1:91,2] = PR[GP1:90,2] + -0.026;
   1:L PR[91] 10mm/sec CNT100;
   1:  PR[GP1:91,1] = PR[GP1:90,1] + -73.394;
   1:  PR[GP1:91,2] = PR[GP1:90,2] + -6.084;
   1:L PR[91] 10mm/sec CNT100;
   1:  PR[GP1:91,1] = PR[GP1:90,1] + -73.300;
   1:  PR[GP1:91,2] = PR[GP1:90,2] + -6.648;
   1:L PR[91] 10mm/sec CNT100;
   1:  PR[GP1:91,1] = PR[GP1:90,1] + -71.617;
   1:  PR[GP1:91,2] = PR[GP1:90,2] + -12.492;
   1:L PR[91] 10mm/sec CNT100;
   1:  PR[GP1:91,1] = PR[GP1:90,1] + -68.866;
   1:  PR[GP1:91,2] = PR[GP1:90,2] + -17.943;
   1:L PR[91] 10mm/sec CNT100;
   1:  PR[GP1:91,1] = PR[GP1:90,1] + -68.582;
   1:  PR[GP1:91,2] = PR[GP1:90,2] + -18.463;
   1:L PR[91] 10mm/sec CNT100;
   1:  PR[GP1:91,1] = PR[GP1:90,1] + -64.896;
   1:  PR[GP1:91,2] = PR[GP1:90,2] + -23.269;
   1:L PR[91] 10mm/sec CNT100;
   1:  PR[GP1:91,1] = PR[GP1:90,1] + -59.893;
   1:  PR[GP1:91,2] = PR[GP1:90,2] + -27.751;
   1:L PR[91] 10mm/sec CNT100;
   1:  PR[GP1:91,1] = PR[GP1:90,1] + -54.732;
   1:  PR[GP1:91,2] = PR[GP1:90,2] + -30.863;
   1:L PR[91] 10mm/sec CNT100;
   1:  PR[GP1:91,1] = PR[GP1:90,1] + -49.014;
   1:  PR[GP1:91,2] = PR[GP1:90,2] + -32.987;
   1:L PR[91] 10mm/sec CNT100;
   1:  PR[GP1:91,1] = PR[GP1:90,1] + -48.421;
   1:  PR[GP1:91,2] = PR[GP1:90,2] + -33.244;
   1:L PR[91] 10mm/sec CNT100;
   1:  PR[GP1:91,1] = PR[GP1:90,1] + -42.496;
   1:  PR[GP1:91,2] = PR[GP1:90,2] + -34.254;
   1:L PR[91] 10mm/sec CNT100;
   1:  PR[GP1:91,1] = PR[GP1:90,1] + -41.772;
   1:  PR[GP1:91,2] = PR[GP1:90,2] + -34.308;
   1:L PR[91] 10mm/sec CNT100;
   1:  PR[GP1:91,1] = PR[GP1:90,1] + -35.782;
   1:  PR[GP1:91,2] = PR[GP1:90,2] + -34.199;
   1:L PR[91] 10mm/sec CNT100;
   1:  PR[GP1:91,1] = PR[GP1:90,1] + -29.904;
   1:  PR[GP1:91,2] = PR[GP1:90,2] + -32.976;
   1:L PR[91] 10mm/sec CNT100;
   1:  PR[GP1:91,1] = PR[GP1:90,1] + -29.144;
   1:  PR[GP1:91,2] = PR[GP1:90,2] + -32.777;
   1:L PR[91] 10mm/sec CNT100;
   1:  PR[GP1:91,1] = PR[GP1:90,1] + -23.657;
   1:  PR[GP1:91,2] = PR[GP1:90,2] + -30.509;
   1:L PR[91] 10mm/sec CNT100;
   1:  PR[GP1:91,1] = PR[GP1:90,1] + -17.946;
   1:  PR[GP1:91,2] = PR[GP1:90,2] + -26.768;
   1:L PR[91] 10mm/sec CNT100;
   1:  PR[GP1:91,1] = PR[GP1:90,1] + -13.708;
   1:  PR[GP1:91,2] = PR[GP1:90,2] + -22.692;
   1:L PR[91] 10mm/sec CNT100;
   1:  PR[GP1:91,1] = PR[GP1:90,1] + -10.263;
   1:  PR[GP1:91,2] = PR[GP1:90,2] + -17.845;
   1:L PR[91] 10mm/sec CNT100;
   1:  PR[GP1:91,1] = PR[GP1:90,1] + -9.708;
   1:  PR[GP1:91,2] = PR[GP1:90,2] + -17.120;
   1:L PR[91] 10mm/sec CNT100;
   1:  PR[GP1:91,1] = PR[GP1:90,1] + -7.262;
   1:  PR[GP1:91,2] = PR[GP1:90,2] + -11.799;
   1:L PR[91] 10mm/sec CNT100;
   1:  PR[GP1:91,1] = PR[GP1:90,1] + -6.949;
   1:  PR[GP1:91,2] = PR[GP1:90,2] + -10.854;
   1:L PR[91] 10mm/sec CNT100;
   1:  PR[GP1:91,1] = PR[GP1:90,1] + -5.630;
   1:  PR[GP1:91,2] = PR[GP1:90,2] + -5.558;
   1:L PR[91] 10mm/sec CNT100;
   1:  PR[GP1:91,1] = PR[GP1:90,1] + -5.768;
   1:  PR[GP1:91,2] = PR[GP1:90,2] + -5.478;
   1:L PR[91] 10mm/sec CNT100;
   1:  PR[GP1:91,1] = PR[GP1:90,1] + -3.816;
   1:  PR[GP1:91,2] = PR[GP1:90,2] + -1.937;
   1:L PR[91] 10mm/sec CNT100;
   1:  PR[GP1:91,1] = PR[GP1:90,1] + -3.655;
   1:  PR[GP1:91,2] = PR[GP1:90,2] + -1.762;
   1:L PR[91] 10mm/sec CNT100;
   1:  PR[GP1:91,1] = PR[GP1:90,1] + -3.435;
   1:  PR[GP1:91,2] = PR[GP1:90,2] + -1.610;
   1:L PR[91] 10mm/sec CNT100;
   1:  PR[GP1:91,1] = PR[GP1:90,1] + -0.407;
   1:  PR[GP1:91,2] = PR[GP1:90,2] + -0.488;
   1:L PR[91] 10mm/sec CNT100;
   1:  PR[GP1:91,1] = PR[GP1:90,1] + -0.095;
   1:  PR[GP1:91,2] = PR[GP1:90,2] + -0.404;
   1:L PR[91] 10mm/sec CNT100;
   1:  PR[GP1:91,1] = PR[GP1:90,1] + 0.946;
   1:L PR[91] 10mm/sec CNT100;
   1:  PR[GP1:91,1] = PR[GP1:90,1] + 4.493;
   1:  PR[GP1:91,2] = PR[GP1:90,2] + -1.729;
   1:L PR[91] 10mm/sec CNT100;
   1:  PR[GP1:91,1] = PR[GP1:90,1] + 6.111;
   1:  PR[GP1:91,2] = PR[GP1:90,2] + -4.651;
   1:L PR[91] 10mm/sec CNT100;
   1:  PR[GP1:91,1] = PR[GP1:90,1] + 6.622;
   1:  PR[GP1:91,2] = PR[GP1:90,2] + -5.466;
   1:L PR[91] 10mm/sec CNT100;
   1:  PR[GP1:91,1] = PR[GP1:90,1] + 6.452;
   1:  PR[GP1:91,2] = PR[GP1:90,2] + -5.563;
   1:L PR[91] 10mm/sec CNT100;
   1:  PR[GP1:91,1] = PR[GP1:90,1] + 7.769;
   1:  PR[GP1:91,2] = PR[GP1:90,2] + -10.855;
   1:L PR[91] 10mm/sec CNT100;
   1:  PR[GP1:91,1] = PR[GP1:90,1] + 8.082;
   1:  PR[GP1:91,2] = PR[GP1:90,2] + -11.799;
   1:L PR[91] 10mm/sec CNT100;
   1:  PR[GP1:91,1] = PR[GP1:90,1] + 10.533;
   1:  PR[GP1:91,2] = PR[GP1:90,2] + -17.129;
   1:L PR[91] 10mm/sec CNT100;
   1:  PR[GP1:91,1] = PR[GP1:90,1] + 13.945;
   1:  PR[GP1:91,2] = PR[GP1:90,2] + -21.930;
   1:L PR[91] 10mm/sec CNT100;
   1:  PR[GP1:91,1] = PR[GP1:90,1] + 14.522;
   1:  PR[GP1:91,2] = PR[GP1:90,2] + -22.685;
   1:L PR[91] 10mm/sec CNT100;
   1:  PR[GP1:91,1] = PR[GP1:90,1] + 18.767;
   1:  PR[GP1:91,2] = PR[GP1:90,2] + -26.768;
   1:L PR[91] 10mm/sec CNT100;
   1:  PR[GP1:91,1] = PR[GP1:90,1] + 24.478;
   1:  PR[GP1:91,2] = PR[GP1:90,2] + -30.509;
   1:L PR[91] 10mm/sec CNT100;
   1:  PR[GP1:91,1] = PR[GP1:90,1] + 29.950;
   1:  PR[GP1:91,2] = PR[GP1:90,2] + -32.771;
   1:L PR[91] 10mm/sec CNT100;
   1:  PR[GP1:91,1] = PR[GP1:90,1] + 35.817;
   1:  PR[GP1:91,2] = PR[GP1:90,2] + -33.992;
   1:L PR[91] 10mm/sec CNT100;
   1:  PR[GP1:91,1] = PR[GP1:90,1] + 36.617;
   1:  PR[GP1:91,2] = PR[GP1:90,2] + -34.199;
   1:L PR[91] 10mm/sec CNT100;
   1:  PR[GP1:91,1] = PR[GP1:90,1] + 42.592;
   1:  PR[GP1:91,2] = PR[GP1:90,2] + -34.308;
   1:L PR[91] 10mm/sec CNT100;
   1:  PR[GP1:91,1] = PR[GP1:90,1] + 43.316;
   1:  PR[GP1:91,2] = PR[GP1:90,2] + -34.254;
   1:L PR[91] 10mm/sec CNT100;
   1:  PR[GP1:91,1] = PR[GP1:90,1] + 49.258;
   1:  PR[GP1:91,2] = PR[GP1:90,2] + -33.241;
   1:L PR[91] 10mm/sec CNT100;
   1:  PR[GP1:91,1] = PR[GP1:90,1] + 54.919;
   1:  PR[GP1:91,2] = PR[GP1:90,2] + -31.138;
   1:L PR[91] 10mm/sec CNT100;
   1:  PR[GP1:91,1] = PR[GP1:90,1] + 55.539;
   1:  PR[GP1:91,2] = PR[GP1:90,2] + -30.871;
   1:L PR[91] 10mm/sec CNT100;
   1:  PR[GP1:91,1] = PR[GP1:90,1] + 60.714;
   1:  PR[GP1:91,2] = PR[GP1:90,2] + -27.751;
   1:L PR[91] 10mm/sec CNT100;
   1:  PR[GP1:91,1] = PR[GP1:90,1] + 65.716;
   1:  PR[GP1:91,2] = PR[GP1:90,2] + -23.269;
   1:L PR[91] 10mm/sec CNT100;
   1:  PR[GP1:91,1] = PR[GP1:90,1] + 69.397;
   1:  PR[GP1:91,2] = PR[GP1:90,2] + -18.470;
   1:L PR[91] 10mm/sec CNT100;
   1:  PR[GP1:91,1] = PR[GP1:90,1] + 72.151;
   1:  PR[GP1:91,2] = PR[GP1:90,2] + -13.012;
   1:L PR[91] 10mm/sec CNT100;
   1:  PR[GP1:91,1] = PR[GP1:90,1] + 72.440;
   1:  PR[GP1:91,2] = PR[GP1:90,2] + -12.483;
   1:L PR[91] 10mm/sec CNT100;
   1:  PR[GP1:91,1] = PR[GP1:90,1] + 74.114;
   1:  PR[GP1:91,2] = PR[GP1:90,2] + -6.669;
   1:L PR[91] 10mm/sec CNT100;
   1:  PR[GP1:91,1] = PR[GP1:90,1] + 74.687;
   1:  PR[GP1:91,2] = PR[GP1:90,2] + -0.559;
   1:L PR[91] 10mm/sec CNT100;
   1:  PR[GP1:91,1] = PR[GP1:90,1] + 74.783;
   1:  PR[GP1:91,2] = PR[GP1:90,2] + 0.017;
   1:L PR[91] 10mm/sec CNT100;
   1:  PR[GP1:91,1] = PR[GP1:90,1] + 74.215;
   1:  PR[GP1:91,2] = PR[GP1:90,2] + 6.075;
   1:L PR[91] 10mm/sec CNT100;
   1:  PR[GP1:91,1] = PR[GP1:90,1] + 74.120;
   1:  PR[GP1:91,2] = PR[GP1:90,2] + 6.639;
   1:L PR[91] 10mm/sec CNT100;
   1:  PR[GP1:91,1] = PR[GP1:90,1] + 72.437;
   1:  PR[GP1:91,2] = PR[GP1:90,2] + 12.483;
   1:L PR[91] 10mm/sec CNT100;
   1:  PR[GP1:91,1] = PR[GP1:90,1] + 69.686;
   1:  PR[GP1:91,2] = PR[GP1:90,2] + 17.935;
   1:L PR[91] 10mm/sec CNT100;
   1:  PR[GP1:91,1] = PR[GP1:90,1] + 69.403;
   1:  PR[GP1:91,2] = PR[GP1:90,2] + 18.453;
   1:L PR[91] 10mm/sec CNT100;
   1:  PR[GP1:91,1] = PR[GP1:90,1] + 65.716;
   1:  PR[GP1:91,2] = PR[GP1:90,2] + 23.260;
   1:L PR[91] 10mm/sec CNT100;
   1:  PR[GP1:91,1] = PR[GP1:90,1] + 60.713;
   1:  PR[GP1:91,2] = PR[GP1:90,2] + 27.742;
   1:L PR[91] 10mm/sec CNT100;
   1:  PR[GP1:91,1] = PR[GP1:90,1] + 55.552;
   1:  PR[GP1:91,2] = PR[GP1:90,2] + 30.854;
   1:L PR[91] 10mm/sec CNT100;
   1:  PR[GP1:91,1] = PR[GP1:90,1] + 49.835;
   1:  PR[GP1:91,2] = PR[GP1:90,2] + 32.978;
   1:L PR[91] 10mm/sec CNT100;
   1:  PR[GP1:91,1] = PR[GP1:90,1] + 49.242;
   1:  PR[GP1:91,2] = PR[GP1:90,2] + 33.235;
   1:L PR[91] 10mm/sec CNT100;
   1:  PR[GP1:91,1] = PR[GP1:90,1] + 43.316;
   1:  PR[GP1:91,2] = PR[GP1:90,2] + 34.245;
   1:L PR[91] 10mm/sec CNT100;
   1:  PR[GP1:91,1] = PR[GP1:90,1] + 42.592;
   1:  PR[GP1:91,2] = PR[GP1:90,2] + 34.299;
   1:L PR[91] 10mm/sec CNT100;
   1:  PR[GP1:91,1] = PR[GP1:90,1] + 36.602;
   1:  PR[GP1:91,2] = PR[GP1:90,2] + 34.190;
   1:L PR[91] 10mm/sec CNT100;
   1:  PR[GP1:91,1] = PR[GP1:90,1] + 30.724;
   1:  PR[GP1:91,2] = PR[GP1:90,2] + 32.967;
   1:L PR[91] 10mm/sec CNT100;
   1:  PR[GP1:91,1] = PR[GP1:90,1] + 29.964;
   1:  PR[GP1:91,2] = PR[GP1:90,2] + 32.768;
   1:L PR[91] 10mm/sec CNT100;
   1:  PR[GP1:91,1] = PR[GP1:90,1] + 24.478;
   1:  PR[GP1:91,2] = PR[GP1:90,2] + 30.500;
   1:L PR[91] 10mm/sec CNT100;
   1:  PR[GP1:91,1] = PR[GP1:90,1] + 18.767;
   1:  PR[GP1:91,2] = PR[GP1:90,2] + 26.759;
   1:L PR[91] 10mm/sec CNT100;
   1:  PR[GP1:91,1] = PR[GP1:90,1] + 14.529;
   1:  PR[GP1:91,2] = PR[GP1:90,2] + 22.683;
   1:L PR[91] 10mm/sec CNT100;
   1:  PR[GP1:91,1] = PR[GP1:90,1] + 11.084;
   1:  PR[GP1:91,2] = PR[GP1:90,2] + 17.836;
   1:L PR[91] 10mm/sec CNT100;
   1:  PR[GP1:91,1] = PR[GP1:90,1] + 10.529;
   1:  PR[GP1:91,2] = PR[GP1:90,2] + 17.111;
   1:L PR[91] 10mm/sec CNT100;
   1:  PR[GP1:91,1] = PR[GP1:90,1] + 8.082;
   1:  PR[GP1:91,2] = PR[GP1:90,2] + 11.790;
   1:L PR[91] 10mm/sec CNT100;
   1:  PR[GP1:91,1] = PR[GP1:90,1] + 7.769;
   1:  PR[GP1:91,2] = PR[GP1:90,2] + 10.845;
   1:L PR[91] 10mm/sec CNT100;
   1:  PR[GP1:91,1] = PR[GP1:90,1] + 6.451;
   1:  PR[GP1:91,2] = PR[GP1:90,2] + 5.551;
   1:L PR[91] 10mm/sec CNT100;
   1:  PR[GP1:91,1] = PR[GP1:90,1] + 6.590;
   1:  PR[GP1:91,2] = PR[GP1:90,2] + 5.471;
   1:L PR[91] 10mm/sec CNT100;
   1:  PR[GP1:91,1] = PR[GP1:90,1] + 4.637;
   1:  PR[GP1:91,2] = PR[GP1:90,2] + 1.928;
   1:L PR[91] 10mm/sec CNT100;
   1:  PR[GP1:91,1] = PR[GP1:90,1] + 4.476;
   1:  PR[GP1:91,2] = PR[GP1:90,2] + 1.754;
   1:L PR[91] 10mm/sec CNT100;
   1:  PR[GP1:91,1] = PR[GP1:90,1] + 4.255;
   1:  PR[GP1:91,2] = PR[GP1:90,2] + 1.601;
   1:L PR[91] 10mm/sec CNT100;
   1:  PR[GP1:91,1] = PR[GP1:90,1] + 1.228;
   1:  PR[GP1:91,2] = PR[GP1:90,2] + 0.479;
   1:L PR[91] 10mm/sec CNT100;
   1:  PR[GP1:91,1] = PR[GP1:90,1] + 0.916;
   1:  PR[GP1:91,2] = PR[GP1:90,2] + 0.396;
   1:L PR[91] 10mm/sec CNT100;
   1:  PR[GP1:91,1] = PR[GP1:90,1] + -0.125;
   1:L PR[91] 10mm/sec CNT100;
   1:  PR[GP1:91,1] = PR[GP1:90,1] + -1.411;
   1:  PR[GP1:91,2] = PR[GP1:90,2] + 0.892;
   1:  PR[GP1:91,3] = PR[GP1:90,3] + 10.640;
   1:L PR[91] 10mm/sec CNT100;
   1:  PR[GP1:91,1] = PR[GP1:90,1] + -2.231;
   1:  PR[GP1:91,2] = PR[GP1:90,2] + 1.219;
   1:L PR[91] 10mm/sec CNT100;
   1:  PR[GP1:91,1] = PR[GP1:90,1] + -2.304;
   1:  PR[GP1:91,2] = PR[GP1:90,2] + 1.222;
   1:L PR[91] 10mm/sec CNT100;
   1:  PR[GP1:91,1] = PR[GP1:90,1] + -3.577;
   1:  PR[GP1:91,2] = PR[GP1:90,2] + 1.726;
   1:L PR[91] 10mm/sec CNT100;
   1:  PR[GP1:91,1] = PR[GP1:90,1] + -4.852;
   1:  PR[GP1:91,2] = PR[GP1:90,2] + 4.028;
   1:L PR[91] 10mm/sec CNT100;
   1:  PR[GP1:91,1] = PR[GP1:90,1] + -5.750;
   1:  PR[GP1:91,2] = PR[GP1:90,2] + 5.460;
   1:L PR[91] 10mm/sec CNT100;
   1:  PR[GP1:91,1] = PR[GP1:90,1] + -5.535;
   1:  PR[GP1:91,2] = PR[GP1:90,2] + 5.581;
   1:L PR[91] 10mm/sec CNT100;
   1:  PR[GP1:91,1] = PR[GP1:90,1] + -6.552;
   1:  PR[GP1:91,2] = PR[GP1:90,2] + 9.664;
   1:L PR[91] 10mm/sec CNT100;
   1:  PR[GP1:91,1] = PR[GP1:90,1] + -7.547;
   1:  PR[GP1:91,2] = PR[GP1:90,2] + 12.667;
   1:L PR[91] 10mm/sec CNT100;
   1:  PR[GP1:91,1] = PR[GP1:90,1] + -9.501;
   1:  PR[GP1:91,2] = PR[GP1:90,2] + 16.918;
   1:L PR[91] 10mm/sec CNT100;
   1:  PR[GP1:91,1] = PR[GP1:90,1] + -12.224;
   1:  PR[GP1:91,2] = PR[GP1:90,2] + 20.749;
   1:L PR[91] 10mm/sec CNT100;
   1:  PR[GP1:91,1] = PR[GP1:90,1] + -14.058;
   1:  PR[GP1:91,2] = PR[GP1:90,2] + 23.150;
   1:L PR[91] 10mm/sec CNT100;
   1:  PR[GP1:91,1] = PR[GP1:90,1] + -17.499;
   1:  PR[GP1:91,2] = PR[GP1:90,2] + 26.460;
   1:L PR[91] 10mm/sec CNT100;
   1:  PR[GP1:91,1] = PR[GP1:90,1] + -21.535;
   1:  PR[GP1:91,2] = PR[GP1:90,2] + 29.098;
   1:L PR[91] 10mm/sec CNT100;
   1:  PR[GP1:91,1] = PR[GP1:90,1] + -23.907;
   1:  PR[GP1:91,2] = PR[GP1:90,2] + 30.671;
   1:L PR[91] 10mm/sec CNT100;
   1:  PR[GP1:91,1] = PR[GP1:90,1] + -28.426;
   1:  PR[GP1:91,2] = PR[GP1:90,2] + 32.540;
   1:L PR[91] 10mm/sec CNT100;
   1:  PR[GP1:91,1] = PR[GP1:90,1] + -33.285;
   1:  PR[GP1:91,2] = PR[GP1:90,2] + 33.551;
   1:L PR[91] 10mm/sec CNT100;
   1:  PR[GP1:91,1] = PR[GP1:90,1] + -35.847;
   1:  PR[GP1:91,2] = PR[GP1:90,2] + 34.214;
   1:L PR[91] 10mm/sec CNT100;
   1:  PR[GP1:91,1] = PR[GP1:90,1] + -40.879;
   1:  PR[GP1:91,2] = PR[GP1:90,2] + 34.306;
   1:L PR[91] 10mm/sec CNT100;
   1:  PR[GP1:91,1] = PR[GP1:90,1] + -43.211;
   1:  PR[GP1:91,2] = PR[GP1:90,2] + 34.130;
   1:L PR[91] 10mm/sec CNT100;
   1:  PR[GP1:91,1] = PR[GP1:90,1] + -48.294;
   1:  PR[GP1:91,2] = PR[GP1:90,2] + 33.264;
   1:L PR[91] 10mm/sec CNT100;
   1:  PR[GP1:91,1] = PR[GP1:90,1] + -53.140;
   1:  PR[GP1:91,2] = PR[GP1:90,2] + 31.464;
   1:L PR[91] 10mm/sec CNT100;
   1:  PR[GP1:91,1] = PR[GP1:90,1] + -55.144;
   1:  PR[GP1:91,2] = PR[GP1:90,2] + 30.601;
   1:L PR[91] 10mm/sec CNT100;
   1:  PR[GP1:91,1] = PR[GP1:90,1] + -59.624;
   1:  PR[GP1:91,2] = PR[GP1:90,2] + 27.899;
   1:L PR[91] 10mm/sec CNT100;
   1:  PR[GP1:91,1] = PR[GP1:90,1] + -63.551;
   1:  PR[GP1:91,2] = PR[GP1:90,2] + 24.387;
   1:L PR[91] 10mm/sec CNT100;
   1:  PR[GP1:91,1] = PR[GP1:90,1] + -65.071;
   1:  PR[GP1:91,2] = PR[GP1:90,2] + 23.003;
   1:L PR[91] 10mm/sec CNT100;
   1:  PR[GP1:91,1] = PR[GP1:90,1] + -68.284;
   1:  PR[GP1:91,2] = PR[GP1:90,2] + 18.813;
   1:L PR[91] 10mm/sec CNT100;
   1:  PR[GP1:91,1] = PR[GP1:90,1] + -70.692;
   1:  PR[GP1:91,2] = PR[GP1:90,2] + 14.043;
   1:L PR[91] 10mm/sec CNT100;
   1:  PR[GP1:91,1] = PR[GP1:90,1] + -71.631;
   1:  PR[GP1:91,2] = PR[GP1:90,2] + 12.318;
   1:L PR[91] 10mm/sec CNT100;
   1:  PR[GP1:91,1] = PR[GP1:90,1] + -73.099;
   1:  PR[GP1:91,2] = PR[GP1:90,2] + 7.221;
   1:L PR[91] 10mm/sec CNT100;
   1:  PR[GP1:91,1] = PR[GP1:90,1] + -73.602;
   1:  PR[GP1:91,2] = PR[GP1:90,2] + 1.853;
   1:L PR[91] 10mm/sec CNT100;
   1:  PR[GP1:91,1] = PR[GP1:90,1] + -73.916;
   1:  PR[GP1:91,2] = PR[GP1:90,2] + -0.026;
   1:L PR[91] 10mm/sec CNT100;
   1:  PR[GP1:91,1] = PR[GP1:90,1] + -73.415;
   1:  PR[GP1:91,2] = PR[GP1:90,2] + -5.369;
   1:L PR[91] 10mm/sec CNT100;
   1:  PR[GP1:91,1] = PR[GP1:90,1] + -73.105;
   1:  PR[GP1:91,2] = PR[GP1:90,2] + -7.209;
   1:L PR[91] 10mm/sec CNT100;
   1:  PR[GP1:91,1] = PR[GP1:90,1] + -71.629;
   1:  PR[GP1:91,2] = PR[GP1:90,2] + -12.336;
   1:L PR[91] 10mm/sec CNT100;
   1:  PR[GP1:91,1] = PR[GP1:90,1] + -69.214;
   1:  PR[GP1:91,2] = PR[GP1:90,2] + -17.122;
   1:L PR[91] 10mm/sec CNT100;
   1:  PR[GP1:91,1] = PR[GP1:90,1] + -68.290;
   1:  PR[GP1:91,2] = PR[GP1:90,2] + -18.814;
   1:L PR[91] 10mm/sec CNT100;
   1:  PR[GP1:91,1] = PR[GP1:90,1] + -65.073;
   1:  PR[GP1:91,2] = PR[GP1:90,2] + -23.009;
   1:L PR[91] 10mm/sec CNT100;
   1:  PR[GP1:91,1] = PR[GP1:90,1] + -61.095;
   1:  PR[GP1:91,2] = PR[GP1:90,2] + -26.566;
   1:L PR[91] 10mm/sec CNT100;
   1:  PR[GP1:91,1] = PR[GP1:90,1] + -59.621;
   1:  PR[GP1:91,2] = PR[GP1:90,2] + -27.910;
   1:L PR[91] 10mm/sec CNT100;
   1:  PR[GP1:91,1] = PR[GP1:90,1] + -55.157;
   1:  PR[GP1:91,2] = PR[GP1:90,2] + -30.602;
   1:L PR[91] 10mm/sec CNT100;
   1:  PR[GP1:91,1] = PR[GP1:90,1] + -50.201;
   1:  PR[GP1:91,2] = PR[GP1:90,2] + -32.443;
   1:L PR[91] 10mm/sec CNT100;
   1:  PR[GP1:91,1] = PR[GP1:90,1] + -48.278;
   1:  PR[GP1:91,2] = PR[GP1:90,2] + -33.276;
   1:L PR[91] 10mm/sec CNT100;
   1:  PR[GP1:91,1] = PR[GP1:90,1] + -43.211;
   1:  PR[GP1:91,2] = PR[GP1:90,2] + -34.139;
   1:L PR[91] 10mm/sec CNT100;
   1:  PR[GP1:91,1] = PR[GP1:90,1] + -40.879;
   1:  PR[GP1:91,2] = PR[GP1:90,2] + -34.315;
   1:L PR[91] 10mm/sec CNT100;
   1:  PR[GP1:91,1] = PR[GP1:90,1] + -35.833;
   1:  PR[GP1:91,2] = PR[GP1:90,2] + -34.223;
   1:L PR[91] 10mm/sec CNT100;
   1:  PR[GP1:91,1] = PR[GP1:90,1] + -30.879;
   1:  PR[GP1:91,2] = PR[GP1:90,2] + -33.192;
   1:L PR[91] 10mm/sec CNT100;
   1:  PR[GP1:91,1] = PR[GP1:90,1] + -28.440;
   1:  PR[GP1:91,2] = PR[GP1:90,2] + -32.554;
   1:L PR[91] 10mm/sec CNT100;
   1:  PR[GP1:91,1] = PR[GP1:90,1] + -23.905;
   1:  PR[GP1:91,2] = PR[GP1:90,2] + -30.679;
   1:L PR[91] 10mm/sec CNT100;
   1:  PR[GP1:91,1] = PR[GP1:90,1] + -19.765;
   1:  PR[GP1:91,2] = PR[GP1:90,2] + -27.973;
   1:L PR[91] 10mm/sec CNT100;
   1:  PR[GP1:91,1] = PR[GP1:90,1] + -17.501;
   1:  PR[GP1:91,2] = PR[GP1:90,2] + -26.470;
   1:L PR[91] 10mm/sec CNT100;
   1:  PR[GP1:91,1] = PR[GP1:90,1] + -14.066;
   1:  PR[GP1:91,2] = PR[GP1:90,2] + -23.166;
   1:L PR[91] 10mm/sec CNT100;
   1:  PR[GP1:91,1] = PR[GP1:90,1] + -11.267;
   1:  PR[GP1:91,2] = PR[GP1:90,2] + -19.229;
   1:L PR[91] 10mm/sec CNT100;
   1:  PR[GP1:91,1] = PR[GP1:90,1] + -9.496;
   1:  PR[GP1:91,2] = PR[GP1:90,2] + -16.917;
   1:L PR[91] 10mm/sec CNT100;
   1:  PR[GP1:91,1] = PR[GP1:90,1] + -7.547;
   1:  PR[GP1:91,2] = PR[GP1:90,2] + -12.676;
   1:L PR[91] 10mm/sec CNT100;
   1:  PR[GP1:91,1] = PR[GP1:90,1] + -6.552;
   1:  PR[GP1:91,2] = PR[GP1:90,2] + -9.674;
   1:L PR[91] 10mm/sec CNT100;
   1:  PR[GP1:91,1] = PR[GP1:90,1] + -5.533;
   1:  PR[GP1:91,2] = PR[GP1:90,2] + -5.584;
   1:L PR[91] 10mm/sec CNT100;
   1:  PR[GP1:91,1] = PR[GP1:90,1] + -5.702;
   1:  PR[GP1:91,2] = PR[GP1:90,2] + -5.485;
   1:L PR[91] 10mm/sec CNT100;
   1:  PR[GP1:91,1] = PR[GP1:90,1] + -5.093;
   1:  PR[GP1:91,2] = PR[GP1:90,2] + -4.314;
   1:L PR[91] 10mm/sec CNT100;
   1:  PR[GP1:91,1] = PR[GP1:90,1] + -3.865;
   1:  PR[GP1:91,2] = PR[GP1:90,2] + -2.095;
   1:L PR[91] 10mm/sec CNT100;
   1:  PR[GP1:91,1] = PR[GP1:90,1] + -3.569;
   1:  PR[GP1:91,2] = PR[GP1:90,2] + -1.773;
   1:L PR[91] 10mm/sec CNT100;
   1:  PR[GP1:91,1] = PR[GP1:90,1] + -3.134;
   1:  PR[GP1:91,2] = PR[GP1:90,2] + -1.474;
   1:L PR[91] 10mm/sec CNT100;
   1:  PR[GP1:91,1] = PR[GP1:90,1] + -0.784;
   1:  PR[GP1:91,2] = PR[GP1:90,2] + -0.602;
   1:L PR[91] 10mm/sec CNT100;
   1:  PR[GP1:91,1] = PR[GP1:90,1] + -0.041;
   1:  PR[GP1:91,2] = PR[GP1:90,2] + -0.404;
   1:L PR[91] 10mm/sec CNT100;
   1:  PR[GP1:91,1] = PR[GP1:90,1] + 0.893;
   1:L PR[91] 10mm/sec CNT100;
   1:  PR[GP1:91,1] = PR[GP1:90,1] + 2.231;
   1:  PR[GP1:91,2] = PR[GP1:90,2] + -0.900;
   1:L PR[91] 10mm/sec CNT100;
   1:  PR[GP1:91,1] = PR[GP1:90,1] + 3.051;
   1:  PR[GP1:91,2] = PR[GP1:90,2] + -1.228;
   1:L PR[91] 10mm/sec CNT100;
   1:  PR[GP1:91,1] = PR[GP1:90,1] + 3.125;
   1:  PR[GP1:91,2] = PR[GP1:90,2] + -1.231;
   1:L PR[91] 10mm/sec CNT100;
   1:  PR[GP1:91,1] = PR[GP1:90,1] + 4.398;
   1:  PR[GP1:91,2] = PR[GP1:90,2] + -1.735;
   1:L PR[91] 10mm/sec CNT100;
   1:  PR[GP1:91,1] = PR[GP1:90,1] + 5.672;
   1:  PR[GP1:91,2] = PR[GP1:90,2] + -4.037;
   1:L PR[91] 10mm/sec CNT100;
   1:  PR[GP1:91,1] = PR[GP1:90,1] + 6.570;
   1:  PR[GP1:91,2] = PR[GP1:90,2] + -5.467;
